Fanuc TP program (LS listing): ultrahose2.ls

/PROG  ultrahose2
/ATTR
COMMENT	= "19-03-19 19:07:18";
PROG_SIZE	= 0;
DEFAULT_GROUP	= 1, *, *, *, *;
/APPL
    ARC Welding Equipment: 1, *, *, *, *;
/MN
   1:  CALL HOME_ALL;
   1:  UFRAME_NUM = 1;
   1:  UTOOL_NUM = 3;
   1:  COL GUARD ADJUST 150;
   1:  PR[91] = PR[90];
   1:  PR[91,1] = PR[90,1] + -69.984;
   1:  PR[91,2] = PR[90,2] + 18.874;
   1:  PR[91,3] = PR[90,3] + 41.795;
   1:L PR[91] R[100]mm/sec CNT100;
   1:  PR[91,1] = PR[90,1] + -74.342;
   1:  PR[91,2] = PR[90,2] + 17.831;
   1:  PR[91,3] = PR[90,3] + 40.507;
   1:L PR[91] R[100]mm/sec CNT100;
   1:  PR[91,1] = PR[90,1] + -76.453;
   1:  PR[91,2] = PR[90,2] + 16.884;
   1:  PR[91,3] = PR[90,3] + 40.519;
   1:L PR[91] R[100]mm/sec CNT100;
   1:  PR[91,1] = PR[90,1] + -78.325;
   1:  PR[91,2] = PR[90,2] + 16.024;
   1:  PR[91,3] = PR[90,3] + 40.526;
   1:L PR[91] R[100]mm/sec CNT100;
   1:  PR[91,1] = PR[90,1] + -81.808;
   1:  PR[91,2] = PR[90,2] + 13.533;
   1:  PR[91,3] = PR[90,3] + 40.531;
   1:L PR[91] R[100]mm/sec CNT100;
   1:  PR[91,1] = PR[90,1] + -84.645;
   1:  PR[91,2] = PR[90,2] + 10.479;
   1:  PR[91,3] = PR[90,3] + 40.543;
   1:L PR[91] R[100]mm/sec CNT100;
   1:  PR[91,1] = PR[90,1] + -86.743;
   1:  PR[91,2] = PR[90,2] + 6.989;
   1:  PR[91,3] = PR[90,3] + 40.554;
   1:L PR[91] R[100]mm/sec CNT100;
   1:  PR[91,1] = PR[90,1] + -88.027;
   1:  PR[91,2] = PR[90,2] + 3.202;
   1:  PR[91,3] = PR[90,3] + 40.565;
   1:L PR[91] R[100]mm/sec CNT100;
   1:  PR[91,1] = PR[90,1] + -88.458;
   1:  PR[91,2] = PR[90,2] + -0.644;
   1:  PR[91,3] = PR[90,3] + 40.576;
   1:L PR[91] R[100]mm/sec CNT100;
   1:  PR[91,1] = PR[90,1] + -88.450;
   1:  PR[91,2] = PR[90,2] + -0.687;
   1:  PR[91,3] = PR[90,3] + 40.586;
   1:L PR[91] R[100]mm/sec CNT100;
   1:  PR[91,1] = PR[90,1] + -88.230;
   1:  PR[91,2] = PR[90,2] + -1.609;
   1:L PR[91] R[100]mm/sec CNT100;
   1:  PR[91,1] = PR[90,1] + -87.903;
   1:  PR[91,2] = PR[90,2] + -4.678;
   1:  PR[91,3] = PR[90,3] + 40.589;
   1:L PR[91] R[100]mm/sec CNT100;
   1:  PR[91,1] = PR[90,1] + -86.648;
   1:  PR[91,2] = PR[90,2] + -8.471;
   1:  PR[91,3] = PR[90,3] + 40.597;
   1:L PR[91] R[100]mm/sec CNT100;
   1:  PR[91,1] = PR[90,1] + -84.603;
   1:  PR[91,2] = PR[90,2] + -11.959;
   1:  PR[91,3] = PR[90,3] + 40.608;
   1:L PR[91] R[100]mm/sec CNT100;
   1:  PR[91,1] = PR[90,1] + -81.844;
   1:  PR[91,2] = PR[90,2] + -15.001;
   1:  PR[91,3] = PR[90,3] + 40.619;
   1:L PR[91] R[100]mm/sec CNT100;
   1:  PR[91,1] = PR[90,1] + -79.437;
   1:  PR[91,2] = PR[90,2] + -16.759;
   1:  PR[91,3] = PR[90,3] + 40.630;
   1:L PR[91] R[100]mm/sec CNT100;
   1:  PR[91,1] = PR[90,1] + -78.444;
   1:  PR[91,2] = PR[90,2] + -17.461;
   1:  PR[91,3] = PR[90,3] + 40.638;
   1:L PR[91] R[100]mm/sec CNT100;
   1:  PR[91,1] = PR[90,1] + -74.380;
   1:  PR[91,2] = PR[90,2] + -19.282;
   1:  PR[91,3] = PR[90,3] + 40.641;
   1:L PR[91] R[100]mm/sec CNT100;
   1:  PR[91,1] = PR[90,1] + -71.242;
   1:  PR[91,2] = PR[90,2] + -20.012;
   1:  PR[91,3] = PR[90,3] + 40.653;
   1:L PR[91] R[100]mm/sec CNT100;
   1:  PR[91,1] = PR[90,1] + -69.927;
   1:  PR[91,2] = PR[90,2] + -20.339;
   1:  PR[91,3] = PR[90,3] + 40.662;
   1:L PR[91] R[100]mm/sec CNT100;
   1:  PR[91,1] = PR[90,1] + -67.497;
   1:  PR[91,2] = PR[90,2] + -20.438;
   1:  PR[91,3] = PR[90,3] + 40.666;
   1:L PR[91] R[100]mm/sec CNT100;
   1:  PR[91,1] = PR[90,1] + -65.288;
   1:  PR[91,2] = PR[90,2] + -20.565;
   1:  PR[91,3] = PR[90,3] + 40.672;
   1:L PR[91] R[100]mm/sec CNT100;
   1:  PR[91,1] = PR[90,1] + -63.772;
   1:  PR[91,2] = PR[90,2] + -20.339;
   1:  PR[91,3] = PR[90,3] + 40.678;
   1:L PR[91] R[100]mm/sec CNT100;
   1:  PR[91,1] = PR[90,1] + -60.637;
   1:  PR[91,2] = PR[90,2] + -19.928;
   1:  PR[91,3] = PR[90,3] + 40.683;
   1:L PR[91] R[100]mm/sec CNT100;
   1:  PR[91,1] = PR[90,1] + -60.136;
   1:  PR[91,2] = PR[90,2] + -19.751;
   1:  PR[91,3] = PR[90,3] + 40.691;
   1:L PR[91] R[100]mm/sec CNT100;
   1:  PR[91,1] = PR[90,1] + -57.404;
   1:  PR[91,2] = PR[90,2] + -18.836;
   1:  PR[91,3] = PR[90,3] + 40.692;
   1:L PR[91] R[100]mm/sec CNT100;
   1:  PR[91,1] = PR[90,1] + -56.091;
   1:  PR[91,2] = PR[90,2] + -18.448;
   1:  PR[91,3] = PR[90,3] + 40.700;
   1:L PR[91] R[100]mm/sec CNT100;
   1:  PR[91,1] = PR[90,1] + -55.744;
   1:  PR[91,2] = PR[90,2] + -18.304;
   1:  PR[91,3] = PR[90,3] + 40.704;
   1:L PR[91] R[100]mm/sec CNT100;
   1:  PR[91,1] = PR[90,1] + -52.168;
   1:  PR[91,2] = PR[90,2] + -16.450;
   1:  PR[91,3] = PR[90,3] + 40.705;
   1:L PR[91] R[100]mm/sec CNT100;
   1:  PR[91,1] = PR[90,1] + -50.349;
   1:  PR[91,2] = PR[90,2] + -15.196;
   1:  PR[91,3] = PR[90,3] + 40.716;
   1:L PR[91] R[100]mm/sec CNT100;
   1:  PR[91,1] = PR[90,1] + -48.605;
   1:  PR[91,2] = PR[90,2] + -13.769;
   1:  PR[91,3] = PR[90,3] + 40.722;
   1:L PR[91] R[100]mm/sec CNT100;
   1:  PR[91,1] = PR[90,1] + -46.020;
   1:  PR[91,2] = PR[90,2] + -10.909;
   1:  PR[91,3] = PR[90,3] + 40.728;
   1:L PR[91] R[100]mm/sec CNT100;
   1:  PR[91,1] = PR[90,1] + -45.612;
   1:  PR[91,2] = PR[90,2] + -10.381;
   1:  PR[91,3] = PR[90,3] + 40.738;
   1:L PR[91] R[100]mm/sec CNT100;
   1:  PR[91,1] = PR[90,1] + -43.653;
   1:  PR[91,2] = PR[90,2] + -6.601;
   1:  PR[91,3] = PR[90,3] + 40.740;
   1:L PR[91] R[100]mm/sec CNT100;
   1:  PR[91,1] = PR[90,1] + -41.214;
   1:  PR[91,2] = PR[90,2] + -2.508;
   1:  PR[91,3] = PR[90,3] + 40.752;
   1:L PR[91] R[100]mm/sec CNT100;
   1:  PR[91,1] = PR[90,1] + -38.826;
   1:  PR[91,2] = PR[90,2] + -8.659;
   1:  PR[91,3] = PR[90,3] + 40.765;
   1:L PR[91] R[100]mm/sec CNT100;
   1:  PR[91,1] = PR[90,1] + -38.172;
   1:  PR[91,2] = PR[90,2] + -9.871;
   1:  PR[91,3] = PR[90,3] + 40.782;
   1:L PR[91] R[100]mm/sec CNT100;
   1:  PR[91,1] = PR[90,1] + -36.807;
   1:  PR[91,2] = PR[90,2] + -12.023;
   1:  PR[91,3] = PR[90,3] + 40.786;
   1:L PR[91] R[100]mm/sec CNT100;
   1:  PR[91,1] = PR[90,1] + -36.440;
   1:  PR[91,2] = PR[90,2] + -12.526;
   1:  PR[91,3] = PR[90,3] + 40.793;
   1:L PR[91] R[100]mm/sec CNT100;
   1:  PR[91,1] = PR[90,1] + -35.020;
   1:  PR[91,2] = PR[90,2] + -14.098;
   1:  PR[91,3] = PR[90,3] + 40.795;
   1:L PR[91] R[100]mm/sec CNT100;
   1:  PR[91,1] = PR[90,1] + -33.375;
   1:  PR[91,2] = PR[90,2] + -15.749;
   1:  PR[91,3] = PR[90,3] + 40.800;
   1:L PR[91] R[100]mm/sec CNT100;
   1:  PR[91,1] = PR[90,1] + -31.415;
   1:  PR[91,2] = PR[90,2] + -17.146;
   1:  PR[91,3] = PR[90,3] + 40.807;
   1:L PR[91] R[100]mm/sec CNT100;
   1:  PR[91,1] = PR[90,1] + -29.729;
   1:  PR[91,2] = PR[90,2] + -18.223;
   1:  PR[91,3] = PR[90,3] + 40.813;
   1:L PR[91] R[100]mm/sec CNT100;
   1:  PR[91,1] = PR[90,1] + -27.094;
   1:  PR[91,2] = PR[90,2] + -19.351;
   1:  PR[91,3] = PR[90,3] + 40.819;
   1:L PR[91] R[100]mm/sec CNT100;
   1:  PR[91,1] = PR[90,1] + -25.614;
   1:  PR[91,2] = PR[90,2] + -19.892;
   1:  PR[91,3] = PR[90,3] + 40.826;
   1:L PR[91] R[100]mm/sec CNT100;
   1:  PR[91,1] = PR[90,1] + -22.266;
   1:  PR[91,2] = PR[90,2] + -20.539;
   1:  PR[91,3] = PR[90,3] + 40.831;
   1:L PR[91] R[100]mm/sec CNT100;
   1:  PR[91,1] = PR[90,1] + -21.213;
   1:  PR[91,2] = PR[90,2] + -20.681;
   1:  PR[91,3] = PR[90,3] + 40.840;
   1:L PR[91] R[100]mm/sec CNT100;
   1:  PR[91,1] = PR[90,1] + -17.203;
   1:  PR[91,2] = PR[90,2] + -20.585;
   1:  PR[91,3] = PR[90,3] + 40.843;
   1:L PR[91] R[100]mm/sec CNT100;
   1:  PR[91,1] = PR[90,1] + -16.723;
   1:  PR[91,2] = PR[90,2] + -20.545;
   1:  PR[91,3] = PR[90,3] + 40.853;
   1:L PR[91] R[100]mm/sec CNT100;
   1:  PR[91,1] = PR[90,1] + -12.288;
   1:  PR[91,2] = PR[90,2] + -19.457;
   1:  PR[91,3] = PR[90,3] + 40.855;
   1:L PR[91] R[100]mm/sec CNT100;
   1:  PR[91,1] = PR[90,1] + -11.843;
   1:  PR[91,2] = PR[90,2] + -19.237;
   1:  PR[91,3] = PR[90,3] + 40.867;
   1:L PR[91] R[100]mm/sec CNT100;
   1:  PR[91,1] = PR[90,1] + -8.024;
   1:  PR[91,2] = PR[90,2] + -17.468;
   1:  PR[91,3] = PR[90,3] + 40.868;
   1:L PR[91] R[100]mm/sec CNT100;
   1:  PR[91,1] = PR[90,1] + -7.652;
   1:  PR[91,2] = PR[90,2] + -17.222;
   1:  PR[91,3] = PR[90,3] + 40.880;
   1:L PR[91] R[100]mm/sec CNT100;
   1:  PR[91,1] = PR[90,1] + -4.356;
   1:  PR[91,2] = PR[90,2] + -14.690;
   1:  PR[91,3] = PR[90,3] + 40.881;
   1:L PR[91] R[100]mm/sec CNT100;
   1:  PR[91,1] = PR[90,1] + -3.570;
   1:  PR[91,2] = PR[90,2] + -13.848;
   1:  PR[91,3] = PR[90,3] + 40.892;
   1:L PR[91] R[100]mm/sec CNT100;
   1:  PR[91,1] = PR[90,1] + -1.393;
   1:  PR[91,2] = PR[90,2] + -11.178;
   1:  PR[91,3] = PR[90,3] + 40.895;
   1:L PR[91] R[100]mm/sec CNT100;
   1:  PR[91,1] = PR[90,1] + -0.641;
   1:  PR[91,2] = PR[90,2] + -9.753;
   1:  PR[91,3] = PR[90,3] + 40.905;
   1:L PR[91] R[100]mm/sec CNT100;
   1:  PR[91,1] = PR[90,1] + 0.012;
   1:  PR[91,2] = PR[90,2] + -8.375;
   1:  PR[91,3] = PR[90,3] + 40.909;
   1:L PR[91] R[100]mm/sec CNT100;
   1:  PR[91,1] = PR[90,1] + 2.040;
   1:  PR[91,2] = PR[90,2] + -2.988;
   1:  PR[91,3] = PR[90,3] + 40.913;
   1:L PR[91] R[100]mm/sec CNT100;
   1:  PR[91,1] = PR[90,1] + 4.720;
   1:  PR[91,2] = PR[90,2] + -9.678;
   1:  PR[91,3] = PR[90,3] + 40.929;
   1:L PR[91] R[100]mm/sec CNT100;
   1:  PR[91,1] = PR[90,1] + 5.572;
   1:  PR[91,2] = PR[90,2] + -11.376;
   1:  PR[91,3] = PR[90,3] + 40.948;
   1:L PR[91] R[100]mm/sec CNT100;
   1:  PR[91,1] = PR[90,1] + 7.346;
   1:  PR[91,2] = PR[90,2] + -13.668;
   1:  PR[91,3] = PR[90,3] + 40.953;
   1:L PR[91] R[100]mm/sec CNT100;
   1:  PR[91,1] = PR[90,1] + 7.981;
   1:  PR[91,2] = PR[90,2] + -14.582;
   1:  PR[91,3] = PR[90,3] + 40.961;
   1:L PR[91] R[100]mm/sec CNT100;
   1:  PR[91,1] = PR[90,1] + 9.322;
   1:  PR[91,2] = PR[90,2] + -15.995;
   1:  PR[91,3] = PR[90,3] + 40.964;
   1:L PR[91] R[100]mm/sec CNT100;
   1:  PR[91,1] = PR[90,1] + 12.105;
   1:  PR[91,2] = PR[90,2] + -18.105;
   1:  PR[91,3] = PR[90,3] + 40.969;
   1:L PR[91] R[100]mm/sec CNT100;
   1:  PR[91,1] = PR[90,1] + 13.658;
   1:  PR[91,2] = PR[90,2] + -19.073;
   1:  PR[91,3] = PR[90,3] + 40.979;
   1:L PR[91] R[100]mm/sec CNT100;
   1:  PR[91,1] = PR[90,1] + 17.034;
   1:  PR[91,2] = PR[90,2] + -20.451;
   1:  PR[91,3] = PR[90,3] + 40.984;
   1:L PR[91] R[100]mm/sec CNT100;
   1:  PR[91,1] = PR[90,1] + 18.629;
   1:  PR[91,2] = PR[90,2] + -20.956;
   1:  PR[91,3] = PR[90,3] + 40.994;
   1:L PR[91] R[100]mm/sec CNT100;
   1:  PR[91,1] = PR[90,1] + 22.409;
   1:  PR[91,2] = PR[90,2] + -21.441;
   1:  PR[91,3] = PR[90,3] + 40.998;
   1:L PR[91] R[100]mm/sec CNT100;
   1:  PR[91,1] = PR[90,1] + 23.913;
   1:  PR[91,2] = PR[90,2] + -21.527;
   1:  PR[91,3] = PR[90,3] + 41.008;
   1:L PR[91] R[100]mm/sec CNT100;
   1:  PR[91,1] = PR[90,1] + 27.852;
   1:  PR[91,2] = PR[90,2] + -21.002;
   1:  PR[91,3] = PR[90,3] + 41.012;
   1:L PR[91] R[100]mm/sec CNT100;
   1:  PR[91,1] = PR[90,1] + 29.169;
   1:  PR[91,2] = PR[90,2] + -20.747;
   1:  PR[91,3] = PR[90,3] + 41.023;
   1:L PR[91] R[100]mm/sec CNT100;
   1:  PR[91,1] = PR[90,1] + 32.982;
   1:  PR[91,2] = PR[90,2] + -19.175;
   1:  PR[91,3] = PR[90,3] + 41.027;
   1:L PR[91] R[100]mm/sec CNT100;
   1:  PR[91,1] = PR[90,1] + 34.056;
   1:  PR[91,2] = PR[90,2] + -18.671;
   1:  PR[91,3] = PR[90,3] + 41.038;
   1:L PR[91] R[100]mm/sec CNT100;
   1:  PR[91,1] = PR[90,1] + 37.540;
   1:  PR[91,2] = PR[90,2] + -16.026;
   1:  PR[91,3] = PR[90,3] + 41.041;
   1:L PR[91] R[100]mm/sec CNT100;
   1:  PR[91,1] = PR[90,1] + 37.772;
   1:  PR[91,2] = PR[90,2] + -15.879;
   1:  PR[91,3] = PR[90,3] + 41.053;
   1:L PR[91] R[100]mm/sec CNT100;
   1:  PR[91,1] = PR[90,1] + 38.445;
   1:  PR[91,2] = PR[90,2] + -15.255;
   1:  PR[91,3] = PR[90,3] + 41.054;
   1:L PR[91] R[100]mm/sec CNT100;
   1:  PR[91,1] = PR[90,1] + 38.894;
   1:  PR[91,2] = PR[90,2] + -14.763;
   1:  PR[91,3] = PR[90,3] + 41.056;
   1:L PR[91] R[100]mm/sec CNT100;
   1:  PR[91,1] = PR[90,1] + 41.536;
   1:  PR[91,2] = PR[90,2] + -11.574;
   1:  PR[91,3] = PR[90,3] + 41.058;
   1:L PR[91] R[100]mm/sec CNT100;
   1:  PR[91,1] = PR[90,1] + 44.233;
   1:  PR[91,2] = PR[90,2] + -14.310;
   1:  PR[91,3] = PR[90,3] + 41.069;
   1:L PR[91] R[100]mm/sec CNT100;
   1:  PR[91,1] = PR[90,1] + 46.319;
   1:  PR[91,2] = PR[90,2] + -15.800;
   1:  PR[91,3] = PR[90,3] + 41.080;
   1:L PR[91] R[100]mm/sec CNT100;
   1:  PR[91,1] = PR[90,1] + 49.840;
   1:  PR[91,2] = PR[90,2] + -18.103;
   1:  PR[91,3] = PR[90,3] + 41.086;
   1:L PR[91] R[100]mm/sec CNT100;
   1:  PR[91,1] = PR[90,1] + 50.344;
   1:  PR[91,2] = PR[90,2] + -18.304;
   1:  PR[91,3] = PR[90,3] + 41.098;
   1:L PR[91] R[100]mm/sec CNT100;
   1:  PR[91,1] = PR[90,1] + 54.403;
   1:  PR[91,2] = PR[90,2] + -20.079;
   1:  PR[91,3] = PR[90,3] + 41.099;
   1:L PR[91] R[100]mm/sec CNT100;
   1:  PR[91,1] = PR[90,1] + 56.501;
   1:  PR[91,2] = PR[90,2] + -20.784;
   1:  PR[91,3] = PR[90,3] + 41.111;
   1:L PR[91] R[100]mm/sec CNT100;
   1:  PR[91,1] = PR[90,1] + 59.032;
   1:  PR[91,2] = PR[90,2] + -21.322;
   1:  PR[91,3] = PR[90,3] + 41.117;
   1:L PR[91] R[100]mm/sec CNT100;
   1:  PR[91,1] = PR[90,1] + 63.968;
   1:  PR[91,2] = PR[90,2] + -21.878;
   1:  PR[91,3] = PR[90,3] + 41.124;
   1:L PR[91] R[100]mm/sec CNT100;
   1:  PR[91,1] = PR[90,1] + 64.084;
   1:  PR[91,2] = PR[90,2] + -21.880;
   1:  PR[91,3] = PR[90,3] + 41.138;
   1:L PR[91] R[100]mm/sec CNT100;
   1:  PR[91,1] = PR[90,1] + 64.736;
   1:  PR[91,2] = PR[90,2] + -21.820;
   1:L PR[91] R[100]mm/sec CNT100;
   1:  PR[91,1] = PR[90,1] + 69.228;
   1:  PR[91,2] = PR[90,2] + -21.507;
   1:  PR[91,3] = PR[90,3] + 41.140;
   1:L PR[91] R[100]mm/sec CNT100;
   1:  PR[91,1] = PR[90,1] + 70.397;
   1:  PR[91,2] = PR[90,2] + -21.313;
   1:  PR[91,3] = PR[90,3] + 41.152;
   1:L PR[91] R[100]mm/sec CNT100;
   1:  PR[91,1] = PR[90,1] + 73.749;
   1:  PR[91,2] = PR[90,2] + -20.328;
   1:  PR[91,3] = PR[90,3] + 41.155;
   1:L PR[91] R[100]mm/sec CNT100;
   1:  PR[91,1] = PR[90,1] + 75.998;
   1:  PR[91,2] = PR[90,2] + -19.468;
   1:  PR[91,3] = PR[90,3] + 41.164;
   1:L PR[91] R[100]mm/sec CNT100;
   1:  PR[91,1] = PR[90,1] + 77.841;
   1:  PR[91,2] = PR[90,2] + -18.450;
   1:  PR[91,3] = PR[90,3] + 41.171;
   1:L PR[91] R[100]mm/sec CNT100;
   1:  PR[91,1] = PR[90,1] + 80.605;
   1:  PR[91,2] = PR[90,2] + -16.678;
   1:  PR[91,3] = PR[90,3] + 41.177;
   1:L PR[91] R[100]mm/sec CNT100;
   1:  PR[91,1] = PR[90,1] + 81.422;
   1:  PR[91,2] = PR[90,2] + -15.949;
   1:  PR[91,3] = PR[90,3] + 41.186;
   1:L PR[91] R[100]mm/sec CNT100;
   1:  PR[91,1] = PR[90,1] + 84.184;
   1:  PR[91,2] = PR[90,2] + -13.215;
   1:  PR[91,3] = PR[90,3] + 41.189;
   1:L PR[91] R[100]mm/sec CNT100;
   1:  PR[91,1] = PR[90,1] + 84.403;
   1:  PR[91,2] = PR[90,2] + -12.900;
   1:  PR[91,3] = PR[90,3] + 41.199;
   1:L PR[91] R[100]mm/sec CNT100;
   1:  PR[91,1] = PR[90,1] + 86.719;
   1:  PR[91,2] = PR[90,2] + -9.308;
   1:  PR[91,3] = PR[90,3] + 41.200;
   1:L PR[91] R[100]mm/sec CNT100;
   1:  PR[91,1] = PR[90,1] + 87.451;
   1:  PR[91,2] = PR[90,2] + -7.293;
   1:  PR[91,3] = PR[90,3] + 41.212;
   1:L PR[91] R[100]mm/sec CNT100;
   1:  PR[91,1] = PR[90,1] + 88.212;
   1:  PR[91,2] = PR[90,2] + -5.114;
   1:  PR[91,3] = PR[90,3] + 41.217;
   1:L PR[91] R[100]mm/sec CNT100;
   1:  PR[91,1] = PR[90,1] + 88.706;
   1:  PR[91,2] = PR[90,2] + -0.729;
   1:  PR[91,3] = PR[90,3] + 41.224;
   1:L PR[91] R[100]mm/sec CNT100;
   1:  PR[91,1] = PR[90,1] + 88.212;
   1:  PR[91,2] = PR[90,2] + 3.655;
   1:  PR[91,3] = PR[90,3] + 41.236;
   1:L PR[91] R[100]mm/sec CNT100;
   1:  PR[91,1] = PR[90,1] + 87.451;
   1:  PR[91,2] = PR[90,2] + 5.834;
   1:  PR[91,3] = PR[90,3] + 41.247;
   1:L PR[91] R[100]mm/sec CNT100;
   1:  PR[91,1] = PR[90,1] + 86.719;
   1:  PR[91,2] = PR[90,2] + 7.849;
   1:  PR[91,3] = PR[90,3] + 41.254;
   1:L PR[91] R[100]mm/sec CNT100;
   1:  PR[91,1] = PR[90,1] + 84.403;
   1:  PR[91,2] = PR[90,2] + 11.441;
   1:  PR[91,3] = PR[90,3] + 41.259;
   1:L PR[91] R[100]mm/sec CNT100;
   1:  PR[91,1] = PR[90,1] + 84.184;
   1:  PR[91,2] = PR[90,2] + 11.756;
   1:  PR[91,3] = PR[90,3] + 41.271;
   1:L PR[91] R[100]mm/sec CNT100;
   1:  PR[91,1] = PR[90,1] + 81.422;
   1:  PR[91,2] = PR[90,2] + 14.490;
   1:  PR[91,3] = PR[90,3] + 41.272;
   1:L PR[91] R[100]mm/sec CNT100;
   1:  PR[91,1] = PR[90,1] + 80.605;
   1:  PR[91,2] = PR[90,2] + 15.219;
   1:  PR[91,3] = PR[90,3] + 41.283;
   1:L PR[91] R[100]mm/sec CNT100;
   1:  PR[91,1] = PR[90,1] + 77.841;
   1:  PR[91,2] = PR[90,2] + 16.991;
   1:  PR[91,3] = PR[90,3] + 41.285;
   1:L PR[91] R[100]mm/sec CNT100;
   1:  PR[91,1] = PR[90,1] + 75.998;
   1:  PR[91,2] = PR[90,2] + 18.009;
   1:  PR[91,3] = PR[90,3] + 41.294;
   1:L PR[91] R[100]mm/sec CNT100;
   1:  PR[91,1] = PR[90,1] + 73.749;
   1:  PR[91,2] = PR[90,2] + 18.869;
   1:  PR[91,3] = PR[90,3] + 41.300;
   1:L PR[91] R[100]mm/sec CNT100;
   1:  PR[91,1] = PR[90,1] + 70.398;
   1:  PR[91,2] = PR[90,2] + 19.854;
   1:  PR[91,3] = PR[90,3] + 41.307;
   1:L PR[91] R[100]mm/sec CNT100;
   1:  PR[91,1] = PR[90,1] + 69.229;
   1:  PR[91,2] = PR[90,2] + 20.048;
   1:  PR[91,3] = PR[90,3] + 41.316;
   1:L PR[91] R[100]mm/sec CNT100;
   1:  PR[91,1] = PR[90,1] + 64.736;
   1:  PR[91,2] = PR[90,2] + 20.362;
   1:  PR[91,3] = PR[90,3] + 41.319;
   1:L PR[91] R[100]mm/sec CNT100;
   1:  PR[91,1] = PR[90,1] + 64.085;
   1:  PR[91,2] = PR[90,2] + 20.421;
   1:  PR[91,3] = PR[90,3] + 41.331;
   1:L PR[91] R[100]mm/sec CNT100;
   1:  PR[91,1] = PR[90,1] + 63.965;
   1:  PR[91,2] = PR[90,2] + 20.419;
   1:  PR[91,3] = PR[90,3] + 41.333;
   1:L PR[91] R[100]mm/sec CNT100;
   1:  PR[91,1] = PR[90,1] + 59.012;
   1:  PR[91,2] = PR[90,2] + 19.862;
   1:L PR[91] R[100]mm/sec CNT100;
   1:  PR[91,1] = PR[90,1] + 56.444;
   1:  PR[91,2] = PR[90,2] + 19.308;
   1:  PR[91,3] = PR[90,3] + 41.347;
   1:L PR[91] R[100]mm/sec CNT100;
   1:  PR[91,1] = PR[90,1] + 54.358;
   1:  PR[91,2] = PR[90,2] + 18.607;
   1:  PR[91,3] = PR[90,3] + 41.354;
   1:L PR[91] R[100]mm/sec CNT100;
   1:  PR[91,1] = PR[90,1] + 50.348;
   1:  PR[91,2] = PR[90,2] + 16.837;
   1:  PR[91,3] = PR[90,3] + 41.360;
   1:L PR[91] R[100]mm/sec CNT100;
   1:  PR[91,1] = PR[90,1] + 49.750;
   1:  PR[91,2] = PR[90,2] + 16.598;
   1:  PR[91,3] = PR[90,3] + 41.372;
   1:L PR[91] R[100]mm/sec CNT100;
   1:  PR[91,1] = PR[90,1] + 46.292;
   1:  PR[91,2] = PR[90,2] + 14.311;
   1:  PR[91,3] = PR[90,3] + 41.374;
   1:L PR[91] R[100]mm/sec CNT100;
   1:  PR[91,1] = PR[90,1] + 44.217;
   1:  PR[91,2] = PR[90,2] + 12.836;
   1:  PR[91,3] = PR[90,3] + 41.385;
   1:L PR[91] R[100]mm/sec CNT100;
   1:  PR[91,1] = PR[90,1] + 41.504;
   1:  PR[91,2] = PR[90,2] + 9.965;
   1:  PR[91,3] = PR[90,3] + 41.392;
   1:L PR[91] R[100]mm/sec CNT100;
   1:  PR[91,1] = PR[90,1] + 38.885;
   1:  PR[91,2] = PR[90,2] + 13.307;
   1:  PR[91,3] = PR[90,3] + 41.402;
   1:L PR[91] R[100]mm/sec CNT100;
   1:  PR[91,1] = PR[90,1] + 37.659;
   1:  PR[91,2] = PR[90,2] + 14.522;
   1:  PR[91,3] = PR[90,3] + 41.414;
   1:L PR[91] R[100]mm/sec CNT100;
   1:  PR[91,1] = PR[90,1] + 34.585;
   1:  PR[91,2] = PR[90,2] + 16.847;
   1:  PR[91,3] = PR[90,3] + 41.418;
   1:L PR[91] R[100]mm/sec CNT100;
   1:  PR[91,1] = PR[90,1] + 34.176;
   1:  PR[91,2] = PR[90,2] + 17.142;
   1:  PR[91,3] = PR[90,3] + 41.429;
   1:L PR[91] R[100]mm/sec CNT100;
   1:  PR[91,1] = PR[90,1] + 34.085;
   1:  PR[91,2] = PR[90,2] + 17.201;
   1:  PR[91,3] = PR[90,3] + 41.430;
   1:L PR[91] R[100]mm/sec CNT100;
   1:  PR[91,1] = PR[90,1] + 32.952;
   1:  PR[91,2] = PR[90,2] + 17.734;
   1:L PR[91] R[100]mm/sec CNT100;
   1:  PR[91,1] = PR[90,1] + 29.141;
   1:  PR[91,2] = PR[90,2] + 19.296;
   1:  PR[91,3] = PR[90,3] + 41.434;
   1:L PR[91] R[100]mm/sec CNT100;
   1:  PR[91,1] = PR[90,1] + 27.825;
   1:  PR[91,2] = PR[90,2] + 19.551;
   1:  PR[91,3] = PR[90,3] + 41.445;
   1:L PR[91] R[100]mm/sec CNT100;
   1:  PR[91,1] = PR[90,1] + 23.890;
   1:  PR[91,2] = PR[90,2] + 20.068;
   1:  PR[91,3] = PR[90,3] + 41.449;
   1:L PR[91] R[100]mm/sec CNT100;
   1:  PR[91,1] = PR[90,1] + 22.387;
   1:  PR[91,2] = PR[90,2] + 19.982;
   1:  PR[91,3] = PR[90,3] + 41.459;
   1:L PR[91] R[100]mm/sec CNT100;
   1:  PR[91,1] = PR[90,1] + 18.613;
   1:  PR[91,2] = PR[90,2] + 19.493;
   1:  PR[91,3] = PR[90,3] + 41.463;
   1:L PR[91] R[100]mm/sec CNT100;
   1:  PR[91,1] = PR[90,1] + 17.018;
   1:  PR[91,2] = PR[90,2] + 18.989;
   1:  PR[91,3] = PR[90,3] + 41.474;
   1:L PR[91] R[100]mm/sec CNT100;
   1:  PR[91,1] = PR[90,1] + 13.648;
   1:  PR[91,2] = PR[90,2] + 17.609;
   1:  PR[91,3] = PR[90,3] + 41.478;
   1:L PR[91] R[100]mm/sec CNT100;
   1:  PR[91,1] = PR[90,1] + 12.096;
   1:  PR[91,2] = PR[90,2] + 16.642;
   1:  PR[91,3] = PR[90,3] + 41.488;
   1:L PR[91] R[100]mm/sec CNT100;
   1:  PR[91,1] = PR[90,1] + 9.318;
   1:  PR[91,2] = PR[90,2] + 14.532;
   1:  PR[91,3] = PR[90,3] + 41.493;
   1:L PR[91] R[100]mm/sec CNT100;
   1:  PR[91,1] = PR[90,1] + 7.941;
   1:  PR[91,2] = PR[90,2] + 13.084;
   1:  PR[91,3] = PR[90,3] + 41.502;
   1:L PR[91] R[100]mm/sec CNT100;
   1:  PR[91,1] = PR[90,1] + 5.848;
   1:  PR[91,2] = PR[90,2] + 10.378;
   1:  PR[91,3] = PR[90,3] + 41.508;
   1:L PR[91] R[100]mm/sec CNT100;
   1:  PR[91,1] = PR[90,1] + 5.791;
   1:  PR[91,2] = PR[90,2] + 10.293;
   1:  PR[91,3] = PR[90,3] + 41.517;
   1:L PR[91] R[100]mm/sec CNT100;
   1:  PR[91,1] = PR[90,1] + 5.693;
   1:  PR[91,2] = PR[90,2] + 10.137;
   1:L PR[91] R[100]mm/sec CNT100;
   1:  PR[91,1] = PR[90,1] + 4.942;
   1:  PR[91,2] = PR[90,2] + 8.700;
   1:  PR[91,3] = PR[90,3] + 41.518;
   1:L PR[91] R[100]mm/sec CNT100;
   1:  PR[91,1] = PR[90,1] + 4.314;
   1:  PR[91,2] = PR[90,2] + 7.197;
   1:  PR[91,3] = PR[90,3] + 41.522;
   1:L PR[91] R[100]mm/sec CNT100;
   1:  PR[91,1] = PR[90,1] + 2.218;
   1:  PR[91,2] = PR[90,2] + 1.901;
   1:  PR[91,3] = PR[90,3] + 41.527;
   1:L PR[91] R[100]mm/sec CNT100;
   1:  PR[91,1] = PR[90,1] + -0.867;
   1:  PR[91,2] = PR[90,2] + 8.750;
   1:  PR[91,3] = PR[90,3] + 41.542;
   1:L PR[91] R[100]mm/sec CNT100;
   1:  PR[91,1] = PR[90,1] + -1.376;
   1:  PR[91,2] = PR[90,2] + 9.695;
   1:  PR[91,3] = PR[90,3] + 41.562;
   1:L PR[91] R[100]mm/sec CNT100;
   1:  PR[91,1] = PR[90,1] + -3.553;
   1:  PR[91,2] = PR[90,2] + 12.368;
   1:  PR[91,3] = PR[90,3] + 41.565;
   1:L PR[91] R[100]mm/sec CNT100;
   1:  PR[91,1] = PR[90,1] + -4.343;
   1:  PR[91,2] = PR[90,2] + 13.219;
   1:  PR[91,3] = PR[90,3] + 41.574;
   1:L PR[91] R[100]mm/sec CNT100;
   1:  PR[91,1] = PR[90,1] + -7.635;
   1:  PR[91,2] = PR[90,2] + 15.753;
   1:  PR[91,3] = PR[90,3] + 41.578;
   1:L PR[91] R[100]mm/sec CNT100;
   1:  PR[91,1] = PR[90,1] + -8.010;
   1:  PR[91,2] = PR[90,2] + 16.001;
   1:  PR[91,3] = PR[90,3] + 41.589;
   1:L PR[91] R[100]mm/sec CNT100;
   1:  PR[91,1] = PR[90,1] + -11.844;
   1:  PR[91,2] = PR[90,2] + 17.780;
   1:  PR[91,3] = PR[90,3] + 41.590;
   1:L PR[91] R[100]mm/sec CNT100;
   1:  PR[91,1] = PR[90,1] + -12.274;
   1:  PR[91,2] = PR[90,2] + 17.993;
   1:  PR[91,3] = PR[90,3] + 41.601;
   1:L PR[91] R[100]mm/sec CNT100;
   1:  PR[91,1] = PR[90,1] + -16.710;
   1:  PR[91,2] = PR[90,2] + 19.085;
   1:  PR[91,3] = PR[90,3] + 41.603;
   1:L PR[91] R[100]mm/sec CNT100;
   1:  PR[91,1] = PR[90,1] + -17.189;
   1:  PR[91,2] = PR[90,2] + 19.124;
   1:  PR[91,3] = PR[90,3] + 41.615;
   1:L PR[91] R[100]mm/sec CNT100;
   1:  PR[91,1] = PR[90,1] + -21.203;
   1:  PR[91,2] = PR[90,2] + 19.223;
   1:  PR[91,3] = PR[90,3] + 41.616;
   1:L PR[91] R[100]mm/sec CNT100;
   1:  PR[91,1] = PR[90,1] + -22.255;
   1:  PR[91,2] = PR[90,2] + 19.081;
   1:  PR[91,3] = PR[90,3] + 41.627;
   1:L PR[91] R[100]mm/sec CNT100;
   1:  PR[91,1] = PR[90,1] + -25.606;
   1:  PR[91,2] = PR[90,2] + 18.436;
   1:  PR[91,3] = PR[90,3] + 41.630;
   1:L PR[91] R[100]mm/sec CNT100;
   1:  PR[91,1] = PR[90,1] + -27.085;
   1:  PR[91,2] = PR[90,2] + 17.895;
   1:  PR[91,3] = PR[90,3] + 41.639;
   1:L PR[91] R[100]mm/sec CNT100;
   1:  PR[91,1] = PR[90,1] + -29.723;
   1:  PR[91,2] = PR[90,2] + 16.767;
   1:  PR[91,3] = PR[90,3] + 41.644;
   1:L PR[91] R[100]mm/sec CNT100;
   1:  PR[91,1] = PR[90,1] + -31.409;
   1:  PR[91,2] = PR[90,2] + 15.691;
   1:  PR[91,3] = PR[90,3] + 41.651;
   1:L PR[91] R[100]mm/sec CNT100;
   1:  PR[91,1] = PR[90,1] + -33.371;
   1:  PR[91,2] = PR[90,2] + 14.294;
   1:  PR[91,3] = PR[90,3] + 41.657;
   1:L PR[91] R[100]mm/sec CNT100;
   1:  PR[91,1] = PR[90,1] + -35.015;
   1:  PR[91,2] = PR[90,2] + 12.643;
   1:  PR[91,3] = PR[90,3] + 41.663;
   1:L PR[91] R[100]mm/sec CNT100;
   1:  PR[91,1] = PR[90,1] + -36.390;
   1:  PR[91,2] = PR[90,2] + 11.125;
   1:  PR[91,3] = PR[90,3] + 41.669;
   1:L PR[91] R[100]mm/sec CNT100;
   1:  PR[91,1] = PR[90,1] + -37.846;
   1:  PR[91,2] = PR[90,2] + 8.812;
   1:  PR[91,3] = PR[90,3] + 41.675;
   1:L PR[91] R[100]mm/sec CNT100;
   1:  PR[91,1] = PR[90,1] + -38.076;
   1:  PR[91,2] = PR[90,2] + 8.534;
   1:  PR[91,3] = PR[90,3] + 41.682;
   1:L PR[91] R[100]mm/sec CNT100;
   1:  PR[91,1] = PR[90,1] + -38.403;
   1:  PR[91,2] = PR[90,2] + 8.035;
   1:  PR[91,3] = PR[90,3] + 41.683;
   1:L PR[91] R[100]mm/sec CNT100;
   1:  PR[91,1] = PR[90,1] + -38.759;
   1:  PR[91,2] = PR[90,2] + 7.344;
   1:  PR[91,3] = PR[90,3] + 41.685;
   1:L PR[91] R[100]mm/sec CNT100;
   1:  PR[91,1] = PR[90,1] + -39.268;
   1:  PR[91,2] = PR[90,2] + 5.891;
   1:  PR[91,3] = PR[90,3] + 41.687;
   1:L PR[91] R[100]mm/sec CNT100;
   1:  PR[91,1] = PR[90,1] + -39.389;
   1:  PR[91,2] = PR[90,2] + 5.694;
   1:  PR[91,3] = PR[90,3] + 41.691;
   1:L PR[91] R[100]mm/sec CNT100;
   1:  PR[91,1] = PR[90,1] + -41.513;
   1:  PR[91,2] = PR[90,2] + 0.383;
   1:  PR[91,3] = PR[90,3] + 41.692;
   1:L PR[91] R[100]mm/sec CNT100;
   1:  PR[91,1] = PR[90,1] + -44.557;
   1:  PR[91,2] = PR[90,2] + 7.369;
   1:  PR[91,3] = PR[90,3] + 41.707;
   1:L PR[91] R[100]mm/sec CNT100;
   1:  PR[91,1] = PR[90,1] + -45.645;
   1:  PR[91,2] = PR[90,2] + 8.862;
   1:  PR[91,3] = PR[90,3] + 41.728;
   1:L PR[91] R[100]mm/sec CNT100;
   1:  PR[91,1] = PR[90,1] + -47.705;
   1:  PR[91,2] = PR[90,2] + 11.387;
   1:  PR[91,3] = PR[90,3] + 41.733;
   1:L PR[91] R[100]mm/sec CNT100;
   1:  PR[91,1] = PR[90,1] + -48.151;
   1:  PR[91,2] = PR[90,2] + 11.764;
   1:  PR[91,3] = PR[90,3] + 41.742;
   1:L PR[91] R[100]mm/sec CNT100;
   1:  PR[91,1] = PR[90,1] + -49.875;
   1:  PR[91,2] = PR[90,2] + 13.098;
   1:  PR[91,3] = PR[90,3] + 41.743;
   1:L PR[91] R[100]mm/sec CNT100;
   1:  PR[91,1] = PR[90,1] + -51.686;
   1:  PR[91,2] = PR[90,2] + 14.649;
   1:  PR[91,3] = PR[90,3] + 41.749;
   1:L PR[91] R[100]mm/sec CNT100;
   1:  PR[91,1] = PR[90,1] + -55.941;
   1:  PR[91,2] = PR[90,2] + 16.976;
   1:  PR[91,3] = PR[90,3] + 41.756;
   1:L PR[91] R[100]mm/sec CNT100;
   1:  PR[91,1] = PR[90,1] + -58.858;
   1:  PR[91,2] = PR[90,2] + 17.920;
   1:  PR[91,3] = PR[90,3] + 41.769;
   1:L PR[91] R[100]mm/sec CNT100;
   1:  PR[91,1] = PR[90,1] + -60.595;
   1:  PR[91,2] = PR[90,2] + 18.463;
   1:  PR[91,3] = PR[90,3] + 41.777;
   1:L PR[91] R[100]mm/sec CNT100;
   1:  PR[91,1] = PR[90,1] + -65.427;
   1:  PR[91,2] = PR[90,2] + 19.085;
   1:  PR[91,3] = PR[90,3] + 41.782;
   1:L PR[91] R[100]mm/sec CNT100;
   1:  PR[91] = PR[90];
   1:  PR[91,1] = PR[90,1] + -67.474;
   1:  PR[91,3] = PR[90,3] + 43.095;
   1:L PR[91] R[100]mm/sec CNT100;
   1:  PR[91,1] = PR[90,1] + -69.465;
   1:  PR[91,2] = PR[90,2] + 18.992;
   1:  PR[91,3] = PR[90,3] + 41.803;
   1:L PR[91] R[100]mm/sec CNT100;
   1:  PR[91,1] = PR[90,1] + -73.840;
   1:  PR[91,2] = PR[90,2] + 17.937;
   1:  PR[91,3] = PR[90,3] + 41.808;
   1:L PR[91] R[100]mm/sec CNT100;
   1:  PR[91,1] = PR[90,1] + -77.850;
   1:  PR[91,2] = PR[90,2] + 16.111;
   1:  PR[91,3] = PR[90,3] + 41.821;
   1:L PR[91] R[100]mm/sec CNT100;
   1:  PR[91,1] = PR[90,1] + -81.344;
   1:  PR[91,2] = PR[90,2] + 13.606;
   1:  PR[91,3] = PR[90,3] + 41.833;
   1:L PR[91] R[100]mm/sec CNT100;
   1:  PR[91,1] = PR[90,1] + -84.191;
   1:  PR[91,2] = PR[90,2] + 10.533;
   1:  PR[91,3] = PR[90,3] + 41.845;
   1:L PR[91] R[100]mm/sec CNT100;
   1:  PR[91,1] = PR[90,1] + -86.296;
   1:  PR[91,2] = PR[90,2] + 7.025;
   1:  PR[91,3] = PR[90,3] + 41.856;
   1:L PR[91] R[100]mm/sec CNT100;
   1:  PR[91,1] = PR[90,1] + -87.585;
   1:  PR[91,2] = PR[90,2] + 3.222;
   1:  PR[91,3] = PR[90,3] + 41.867;
   1:L PR[91] R[100]mm/sec CNT100;
   1:  PR[91,1] = PR[90,1] + -87.989;
   1:  PR[91,2] = PR[90,2] + -0.429;
   1:  PR[91,3] = PR[90,3] + 41.879;
   1:L PR[91] R[100]mm/sec CNT100;
   1:  PR[91,1] = PR[90,1] + -88.046;
   1:  PR[91,2] = PR[90,2] + -0.702;
   1:  PR[91,3] = PR[90,3] + 41.889;
   1:L PR[91] R[100]mm/sec CNT100;
   1:  PR[91,1] = PR[90,1] + -87.939;
   1:  PR[91,2] = PR[90,2] + -1.154;
   1:L PR[91] R[100]mm/sec CNT100;
   1:  PR[91,1] = PR[90,1] + -87.561;
   1:  PR[91,2] = PR[90,2] + -4.693;
   1:  PR[91,3] = PR[90,3] + 41.891;
   1:L PR[91] R[100]mm/sec CNT100;
   1:  PR[91,1] = PR[90,1] + -86.303;
   1:  PR[91,2] = PR[90,2] + -8.501;
   1:  PR[91,3] = PR[90,3] + 41.901;
   1:L PR[91] R[100]mm/sec CNT100;
   1:  PR[91,1] = PR[90,1] + -84.252;
   1:  PR[91,2] = PR[90,2] + -12.004;
   1:  PR[91,3] = PR[90,3] + 41.912;
   1:L PR[91] R[100]mm/sec CNT100;
   1:  PR[91,1] = PR[90,1] + -82.472;
   1:  PR[91,2] = PR[90,2] + -13.969;
   1:  PR[91,3] = PR[90,3] + 41.923;
   1:L PR[91] R[100]mm/sec CNT100;
   1:  PR[91,1] = PR[90,1] + -81.462;
   1:  PR[91,2] = PR[90,2] + -15.043;
   1:  PR[91,3] = PR[90,3] + 41.930;
   1:L PR[91] R[100]mm/sec CNT100;
   1:  PR[91,1] = PR[90,1] + -77.908;
   1:  PR[91,2] = PR[90,2] + -17.555;
   1:  PR[91,3] = PR[90,3] + 41.934;
   1:L PR[91] R[100]mm/sec CNT100;
   1:  PR[91,1] = PR[90,1] + -74.860;
   1:  PR[91,2] = PR[90,2] + -18.913;
   1:  PR[91,3] = PR[90,3] + 41.946;
   1:L PR[91] R[100]mm/sec CNT100;
   1:  PR[91,1] = PR[90,1] + -73.811;
   1:  PR[91,2] = PR[90,2] + -19.397;
   1:  PR[91,3] = PR[90,3] + 41.955;
   1:L PR[91] R[100]mm/sec CNT100;
   1:  PR[91,1] = PR[90,1] + -71.225;
   1:  PR[91,2] = PR[90,2] + -19.999;
   1:  PR[91,3] = PR[90,3] + 41.959;
   1:L PR[91] R[100]mm/sec CNT100;
   1:  PR[91,1] = PR[90,1] + -69.344;
   1:  PR[91,2] = PR[90,2] + -20.467;
   1:  PR[91,3] = PR[90,3] + 41.966;
   1:L PR[91] R[100]mm/sec CNT100;
   1:  PR[91,1] = PR[90,1] + -67.500;
   1:  PR[91,2] = PR[90,2] + -20.542;
   1:  PR[91,3] = PR[90,3] + 41.971;
   1:L PR[91] R[100]mm/sec CNT100;
   1:  PR[91,1] = PR[90,1] + -64.674;
   1:  PR[91,2] = PR[90,2] + -20.705;
   1:  PR[91,3] = PR[90,3] + 41.976;
   1:L PR[91] R[100]mm/sec CNT100;
   1:  PR[91,1] = PR[90,1] + -63.773;
   1:  PR[91,2] = PR[90,2] + -20.570;
   1:  PR[91,3] = PR[90,3] + 41.984;
   1:L PR[91] R[100]mm/sec CNT100;
   1:  PR[91,1] = PR[90,1] + -59.973;
   1:  PR[91,2] = PR[90,2] + -20.073;
   1:  PR[91,3] = PR[90,3] + 41.987;
   1:L PR[91] R[100]mm/sec CNT100;
   1:  PR[91,1] = PR[90,1] + -59.827;
   1:  PR[91,2] = PR[90,2] + -20.023;
   1:  PR[91,3] = PR[90,3] + 41.997;
   1:L PR[91] R[100]mm/sec CNT100;
   1:  PR[91,1] = PR[90,1] + -55.586;
   1:  PR[91,2] = PR[90,2] + -18.768;
   1:  PR[91,3] = PR[90,3] + 41.998;
   1:L PR[91] R[100]mm/sec CNT100;
   1:  PR[91,1] = PR[90,1] + -54.130;
   1:  PR[91,2] = PR[90,2] + -18.165;
   1:  PR[91,3] = PR[90,3] + 42.010;
   1:L PR[91] R[100]mm/sec CNT100;
   1:  PR[91,1] = PR[90,1] + -51.553;
   1:  PR[91,2] = PR[90,2] + -16.829;
   1:  PR[91,3] = PR[90,3] + 42.014;
   1:L PR[91] R[100]mm/sec CNT100;
   1:  PR[91,1] = PR[90,1] + -48.667;
   1:  PR[91,2] = PR[90,2] + -14.840;
   1:  PR[91,3] = PR[90,3] + 42.022;
   1:L PR[91] R[100]mm/sec CNT100;
   1:  PR[91,1] = PR[90,1] + -47.858;
   1:  PR[91,2] = PR[90,2] + -14.177;
   1:  PR[91,3] = PR[90,3] + 42.032;
   1:L PR[91] R[100]mm/sec CNT100;
   1:  PR[91,1] = PR[90,1] + -45.179;
   1:  PR[91,2] = PR[90,2] + -11.215;
   1:  PR[91,3] = PR[90,3] + 42.035;
   1:L PR[91] R[100]mm/sec CNT100;
   1:  PR[91,1] = PR[90,1] + -44.479;
   1:  PR[91,2] = PR[90,2] + -10.536;
   1:  PR[91,3] = PR[90,3] + 42.046;
   1:L PR[91] R[100]mm/sec CNT100;
   1:  PR[91,1] = PR[90,1] + -44.176;
   1:  PR[91,2] = PR[90,2] + -10.050;
   1:  PR[91,3] = PR[90,3] + 42.049;
   1:L PR[91] R[100]mm/sec CNT100;
   1:  PR[91,1] = PR[90,1] + -40.501;
   1:  PR[91,2] = PR[90,2] + -3.883;
   1:  PR[91,3] = PR[90,3] + 42.050;
   1:L PR[91] R[100]mm/sec CNT100;
   1:  PR[91,1] = PR[90,1] + -38.678;
   1:  PR[91,2] = PR[90,2] + -8.579;
   1:  PR[91,3] = PR[90,3] + 42.070;
   1:L PR[91] R[100]mm/sec CNT100;
   1:  PR[91,1] = PR[90,1] + -37.842;
   1:  PR[91,2] = PR[90,2] + -10.127;
   1:  PR[91,3] = PR[90,3] + 42.084;
   1:L PR[91] R[100]mm/sec CNT100;
   1:  PR[91,1] = PR[90,1] + -36.990;
   1:  PR[91,2] = PR[90,2] + -11.484;
   1:  PR[91,3] = PR[90,3] + 42.089;
   1:L PR[91] R[100]mm/sec CNT100;
   1:  PR[91,1] = PR[90,1] + -36.742;
   1:  PR[91,2] = PR[90,2] + -11.857;
   1:  PR[91,3] = PR[90,3] + 42.093;
   1:L PR[91] R[100]mm/sec CNT100;
   1:  PR[91,1] = PR[90,1] + -36.258;
   1:  PR[91,2] = PR[90,2] + -12.520;
   1:  PR[91,3] = PR[90,3] + 42.094;
   1:L PR[91] R[100]mm/sec CNT100;
   1:  PR[91,1] = PR[90,1] + -34.502;
   1:  PR[91,2] = PR[90,2] + -14.463;
   1:  PR[91,3] = PR[90,3] + 42.097;
   1:L PR[91] R[100]mm/sec CNT100;
   1:  PR[91,1] = PR[90,1] + -33.197;
   1:  PR[91,2] = PR[90,2] + -15.773;
   1:  PR[91,3] = PR[90,3] + 42.104;
   1:L PR[91] R[100]mm/sec CNT100;
   1:  PR[91,1] = PR[90,1] + -30.812;
   1:  PR[91,2] = PR[90,2] + -17.474;
   1:  PR[91,3] = PR[90,3] + 42.109;
   1:L PR[91] R[100]mm/sec CNT100;
   1:  PR[91,1] = PR[90,1] + -29.551;
   1:  PR[91,2] = PR[90,2] + -18.279;
   1:  PR[91,3] = PR[90,3] + 42.117;
   1:L PR[91] R[100]mm/sec CNT100;
   1:  PR[91,1] = PR[90,1] + -26.411;
   1:  PR[91,2] = PR[90,2] + -19.623;
   1:  PR[91,3] = PR[90,3] + 42.121;
   1:L PR[91] R[100]mm/sec CNT100;
   1:  PR[91,1] = PR[90,1] + -25.429;
   1:  PR[91,2] = PR[90,2] + -19.982;
   1:  PR[91,3] = PR[90,3] + 42.131;
   1:L PR[91] R[100]mm/sec CNT100;
   1:  PR[91,1] = PR[90,1] + -21.515;
   1:  PR[91,2] = PR[90,2] + -20.738;
   1:  PR[91,3] = PR[90,3] + 42.134;
   1:L PR[91] R[100]mm/sec CNT100;
   1:  PR[91,1] = PR[90,1] + -21.015;
   1:  PR[91,2] = PR[90,2] + -20.806;
   1:  PR[91,3] = PR[90,3] + 42.145;
   1:L PR[91] R[100]mm/sec CNT100;
   1:  PR[91,1] = PR[90,1] + -16.444;
   1:  PR[91,2] = PR[90,2] + -20.690;
   1:  PR[91,3] = PR[90,3] + 42.146;
   1:L PR[91] R[100]mm/sec CNT100;
   1:  PR[91,1] = PR[90,1] + -15.743;
   1:  PR[91,2] = PR[90,2] + -20.518;
   1:  PR[91,3] = PR[90,3] + 42.159;
   1:L PR[91] R[100]mm/sec CNT100;
   1:  PR[91,1] = PR[90,1] + -11.846;
   1:  PR[91,2] = PR[90,2] + -19.653;
   1:  PR[91,3] = PR[90,3] + 42.161;
   1:L PR[91] R[100]mm/sec CNT100;
   1:  PR[91,1] = PR[90,1] + -11.425;
   1:  PR[91,2] = PR[90,2] + -19.495;
   1:  PR[91,3] = PR[90,3] + 42.172;
   1:L PR[91] R[100]mm/sec CNT100;
   1:  PR[91,1] = PR[90,1] + -7.622;
   1:  PR[91,2] = PR[90,2] + -17.734;
   1:  PR[91,3] = PR[90,3] + 42.173;
   1:L PR[91] R[100]mm/sec CNT100;
   1:  PR[91,1] = PR[90,1] + -6.581;
   1:  PR[91,2] = PR[90,2] + -17.046;
   1:  PR[91,3] = PR[90,3] + 42.184;
   1:L PR[91] R[100]mm/sec CNT100;
   1:  PR[91,1] = PR[90,1] + -3.877;
   1:  PR[91,2] = PR[90,2] + -14.968;
   1:  PR[91,3] = PR[90,3] + 42.188;
   1:L PR[91] R[100]mm/sec CNT100;
   1:  PR[91,1] = PR[90,1] + -2.525;
   1:  PR[91,2] = PR[90,2] + -13.518;
   1:  PR[91,3] = PR[90,3] + 42.197;
   1:L PR[91] R[100]mm/sec CNT100;
   1:  PR[91,1] = PR[90,1] + -0.835;
   1:  PR[91,2] = PR[90,2] + -11.446;
   1:  PR[91,3] = PR[90,3] + 42.203;
   1:L PR[91] R[100]mm/sec CNT100;
   1:  PR[91,1] = PR[90,1] + 0.280;
   1:  PR[91,2] = PR[90,2] + -9.333;
   1:  PR[91,3] = PR[90,3] + 42.210;
   1:L PR[91] R[100]mm/sec CNT100;
   1:  PR[91,1] = PR[90,1] + 2.362;
   1:  PR[91,2] = PR[90,2] + -4.651;
   1:  PR[91,3] = PR[90,3] + 42.217;
   1:L PR[91] R[100]mm/sec CNT100;
   1:  PR[91,1] = PR[90,1] + 4.247;
   1:  PR[91,2] = PR[90,2] + -9.356;
   1:  PR[91,3] = PR[90,3] + 42.231;
   1:L PR[91] R[100]mm/sec CNT100;
   1:  PR[91,1] = PR[90,1] + 5.341;
   1:  PR[91,2] = PR[90,2] + -11.537;
   1:  PR[91,3] = PR[90,3] + 42.245;
   1:L PR[91] R[100]mm/sec CNT100;
   1:  PR[91,1] = PR[90,1] + 6.684;
   1:  PR[91,2] = PR[90,2] + -13.272;
   1:  PR[91,3] = PR[90,3] + 42.252;
   1:L PR[91] R[100]mm/sec CNT100;
   1:  PR[91,1] = PR[90,1] + 7.497;
   1:  PR[91,2] = PR[90,2] + -14.443;
   1:  PR[91,3] = PR[90,3] + 42.258;
   1:L PR[91] R[100]mm/sec CNT100;
   1:  PR[91,1] = PR[90,1] + 9.240;
   1:  PR[91,2] = PR[90,2] + -16.279;
   1:  PR[91,3] = PR[90,3] + 42.262;
   1:L PR[91] R[100]mm/sec CNT100;
   1:  PR[91,1] = PR[90,1] + 11.590;
   1:  PR[91,2] = PR[90,2] + -18.061;
   1:  PR[91,3] = PR[90,3] + 42.269;
   1:L PR[91] R[100]mm/sec CNT100;
   1:  PR[91,1] = PR[90,1] + 13.626;
   1:  PR[91,2] = PR[90,2] + -19.330;
   1:  PR[91,3] = PR[90,3] + 42.277;
   1:L PR[91] R[100]mm/sec CNT100;
   1:  PR[91,1] = PR[90,1] + 16.503;
   1:  PR[91,2] = PR[90,2] + -20.505;
   1:  PR[91,3] = PR[90,3] + 42.283;
   1:L PR[91] R[100]mm/sec CNT100;
   1:  PR[91,1] = PR[90,1] + 18.636;
   1:  PR[91,2] = PR[90,2] + -21.180;
   1:  PR[91,3] = PR[90,3] + 42.292;
   1:L PR[91] R[100]mm/sec CNT100;
   1:  PR[91,1] = PR[90,1] + 21.888;
   1:  PR[91,2] = PR[90,2] + -21.597;
   1:  PR[91,3] = PR[90,3] + 42.298;
   1:L PR[91] R[100]mm/sec CNT100;
   1:  PR[91,1] = PR[90,1] + 23.948;
   1:  PR[91,2] = PR[90,2] + -21.715;
   1:  PR[91,3] = PR[90,3] + 42.307;
   1:L PR[91] R[100]mm/sec CNT100;
   1:  PR[91,1] = PR[90,1] + 27.367;
   1:  PR[91,2] = PR[90,2] + -21.260;
   1:  PR[91,3] = PR[90,3] + 42.313;
   1:L PR[91] R[100]mm/sec CNT100;
   1:  PR[91,1] = PR[90,1] + 29.223;
   1:  PR[91,2] = PR[90,2] + -20.900;
   1:  PR[91,3] = PR[90,3] + 42.322;
   1:L PR[91] R[100]mm/sec CNT100;
   1:  PR[91,1] = PR[90,1] + 32.558;
   1:  PR[91,2] = PR[90,2] + -19.525;
   1:  PR[91,3] = PR[90,3] + 42.328;
   1:L PR[91] R[100]mm/sec CNT100;
   1:  PR[91,1] = PR[90,1] + 34.123;
   1:  PR[91,2] = PR[90,2] + -18.790;
   1:  PR[91,3] = PR[90,3] + 42.338;
   1:L PR[91] R[100]mm/sec CNT100;
   1:  PR[91,1] = PR[90,1] + 37.251;
   1:  PR[91,2] = PR[90,2] + -16.417;
   1:  PR[91,3] = PR[90,3] + 42.342;
   1:L PR[91] R[100]mm/sec CNT100;
   1:  PR[91,1] = PR[90,1] + 37.451;
   1:  PR[91,2] = PR[90,2] + -16.306;
   1:  PR[91,3] = PR[90,3] + 42.353;
   1:L PR[91] R[100]mm/sec CNT100;
   1:  PR[91,1] = PR[90,1] + 37.538;
   1:  PR[91,2] = PR[90,2] + -16.247;
   1:  PR[91,3] = PR[90,3] + 42.354;
   1:L PR[91] R[100]mm/sec CNT100;
   1:  PR[91,1] = PR[90,1] + 38.587;
   1:  PR[91,2] = PR[90,2] + -15.273;
   1:L PR[91] R[100]mm/sec CNT100;
   1:  PR[91,1] = PR[90,1] + 39.254;
   1:  PR[91,2] = PR[90,2] + -14.542;
   1:  PR[91,3] = PR[90,3] + 42.358;
   1:L PR[91] R[100]mm/sec CNT100;
   1:  PR[91,1] = PR[90,1] + 40.916;
   1:  PR[91,2] = PR[90,2] + -12.537;
   1:  PR[91,3] = PR[90,3] + 42.361;
   1:L PR[91] R[100]mm/sec CNT100;
   1:  PR[91,1] = PR[90,1] + 42.629;
   1:  PR[91,2] = PR[90,2] + -14.275;
   1:  PR[91,3] = PR[90,3] + 42.368;
   1:L PR[91] R[100]mm/sec CNT100;
   1:  PR[91,1] = PR[90,1] + 45.919;
   1:  PR[91,2] = PR[90,2] + -16.624;
   1:  PR[91,3] = PR[90,3] + 42.375;
   1:L PR[91] R[100]mm/sec CNT100;
   1:  PR[91,1] = PR[90,1] + 48.337;
   1:  PR[91,2] = PR[90,2] + -18.206;
   1:  PR[91,3] = PR[90,3] + 42.386;
   1:L PR[91] R[100]mm/sec CNT100;
   1:  PR[91,1] = PR[90,1] + 49.626;
   1:  PR[91,2] = PR[90,2] + -18.748;
   1:  PR[91,3] = PR[90,3] + 42.394;
   1:L PR[91] R[100]mm/sec CNT100;
   1:  PR[91,1] = PR[90,1] + 52.266;
   1:  PR[91,2] = PR[90,2] + -19.767;
   1:  PR[91,3] = PR[90,3] + 42.398;
   1:L PR[91] R[100]mm/sec CNT100;
   1:  PR[91,1] = PR[90,1] + 54.093;
   1:  PR[91,2] = PR[90,2] + -20.565;
   1:  PR[91,3] = PR[90,3] + 42.406;
   1:L PR[91] R[100]mm/sec CNT100;
   1:  PR[91,1] = PR[90,1] + 54.942;
   1:  PR[91,2] = PR[90,2] + -20.851;
   1:  PR[91,3] = PR[90,3] + 42.411;
   1:L PR[91] R[100]mm/sec CNT100;
   1:  PR[91,1] = PR[90,1] + 58.727;
   1:  PR[91,2] = PR[90,2] + -21.656;
   1:  PR[91,3] = PR[90,3] + 42.414;
   1:L PR[91] R[100]mm/sec CNT100;
   1:  PR[91,1] = PR[90,1] + 62.409;
   1:  PR[91,2] = PR[90,2] + -22.070;
   1:  PR[91,3] = PR[90,3] + 42.424;
   1:L PR[91] R[100]mm/sec CNT100;
   1:  PR[91,1] = PR[90,1] + 63.754;
   1:  PR[91,2] = PR[90,2] + -22.094;
   1:  PR[91,3] = PR[90,3] + 42.434;
   1:L PR[91] R[100]mm/sec CNT100;
   1:  PR[91,1] = PR[90,1] + 67.262;
   1:  PR[91,2] = PR[90,2] + -21.775;
   1:  PR[91,3] = PR[90,3] + 42.438;
   1:L PR[91] R[100]mm/sec CNT100;
   1:  PR[91,1] = PR[90,1] + 69.083;
   1:  PR[91,2] = PR[90,2] + -21.648;
   1:  PR[91,3] = PR[90,3] + 42.448;
   1:L PR[91] R[100]mm/sec CNT100;
   1:  PR[91,1] = PR[90,1] + 69.444;
   1:  PR[91,2] = PR[90,2] + -21.588;
   1:  PR[91,3] = PR[90,3] + 42.453;
   1:L PR[91] R[100]mm/sec CNT100;
   1:  PR[91,1] = PR[90,1] + 73.643;
   1:  PR[91,2] = PR[90,2] + -20.355;
   1:  PR[91,3] = PR[90,3] + 42.454;
   1:L PR[91] R[100]mm/sec CNT100;
   1:  PR[91,1] = PR[90,1] + 75.212;
   1:  PR[91,2] = PR[90,2] + -19.754;
   1:  PR[91,3] = PR[90,3] + 42.466;
   1:L PR[91] R[100]mm/sec CNT100;
   1:  PR[91,1] = PR[90,1] + 77.743;
   1:  PR[91,2] = PR[90,2] + -18.356;
   1:  PR[91,3] = PR[90,3] + 42.471;
   1:L PR[91] R[100]mm/sec CNT100;
   1:  PR[91,1] = PR[90,1] + 79.954;
   1:  PR[91,2] = PR[90,2] + -16.939;
   1:  PR[91,3] = PR[90,3] + 42.479;
   1:L PR[91] R[100]mm/sec CNT100;
   1:  PR[91,1] = PR[90,1] + 81.304;
   1:  PR[91,2] = PR[90,2] + -15.734;
   1:  PR[91,3] = PR[90,3] + 42.486;
   1:L PR[91] R[100]mm/sec CNT100;
   1:  PR[91,1] = PR[90,1] + 83.634;
   1:  PR[91,2] = PR[90,2] + -13.427;
   1:  PR[91,3] = PR[90,3] + 42.491;
   1:L PR[91] R[100]mm/sec CNT100;
   1:  PR[91,1] = PR[90,1] + 84.235;
   1:  PR[91,2] = PR[90,2] + -12.565;
   1:  PR[91,3] = PR[90,3] + 42.500;
   1:L PR[91] R[100]mm/sec CNT100;
   1:  PR[91,1] = PR[90,1] + 86.250;
   1:  PR[91,2] = PR[90,2] + -9.439;
   1:  PR[91,3] = PR[90,3] + 42.503;
   1:L PR[91] R[100]mm/sec CNT100;
   1:  PR[91,1] = PR[90,1] + 86.449;
   1:  PR[91,2] = PR[90,2] + -8.925;
   1:  PR[91,3] = PR[90,3] + 42.513;
   1:L PR[91] R[100]mm/sec CNT100;
   1:  PR[91,1] = PR[90,1] + 87.810;
   1:  PR[91,2] = PR[90,2] + -5.162;
   1:  PR[91,3] = PR[90,3] + 42.515;
   1:L PR[91] R[100]mm/sec CNT100;
   1:  PR[91,1] = PR[90,1] + 88.326;
   1:  PR[91,2] = PR[90,2] + -0.792;
   1:  PR[91,3] = PR[90,3] + 42.526;
   1:L PR[91] R[100]mm/sec CNT100;
   1:  PR[91,1] = PR[90,1] + 88.363;
   1:  PR[91,2] = PR[90,2] + -0.627;
   1:  PR[91,3] = PR[90,3] + 42.538;
   1:L PR[91] R[100]mm/sec CNT100;
   1:  PR[91,1] = PR[90,1] + 88.229;
   1:  PR[91,2] = PR[90,2] + 0.528;
   1:L PR[91] R[100]mm/sec CNT100;
   1:  PR[91,1] = PR[90,1] + 87.815;
   1:  PR[91,2] = PR[90,2] + 3.691;
   1:  PR[91,3] = PR[90,3] + 42.541;
   1:L PR[91] R[100]mm/sec CNT100;
   1:  PR[91,1] = PR[90,1] + 86.449;
   1:  PR[91,2] = PR[90,2] + 7.466;
   1:  PR[91,3] = PR[90,3] + 42.550;
   1:L PR[91] R[100]mm/sec CNT100;
   1:  PR[91,1] = PR[90,1] + 86.251;
   1:  PR[91,2] = PR[90,2] + 7.980;
   1:  PR[91,3] = PR[90,3] + 42.561;
   1:L PR[91] R[100]mm/sec CNT100;
   1:  PR[91,1] = PR[90,1] + 84.235;
   1:  PR[91,2] = PR[90,2] + 11.106;
   1:  PR[91,3] = PR[90,3] + 42.563;
   1:L PR[91] R[100]mm/sec CNT100;
   1:  PR[91,1] = PR[90,1] + 83.634;
   1:  PR[91,2] = PR[90,2] + 11.968;
   1:  PR[91,3] = PR[90,3] + 42.573;
   1:L PR[91] R[100]mm/sec CNT100;
   1:  PR[91,1] = PR[90,1] + 81.304;
   1:  PR[91,2] = PR[90,2] + 14.275;
   1:  PR[91,3] = PR[90,3] + 42.576;
   1:L PR[91] R[100]mm/sec CNT100;
   1:  PR[91,1] = PR[90,1] + 79.954;
   1:  PR[91,2] = PR[90,2] + 15.480;
   1:  PR[91,3] = PR[90,3] + 42.585;
   1:L PR[91] R[100]mm/sec CNT100;
   1:  PR[91,1] = PR[90,1] + 77.744;
   1:  PR[91,2] = PR[90,2] + 16.897;
   1:  PR[91,3] = PR[90,3] + 42.590;
   1:L PR[91] R[100]mm/sec CNT100;
   1:  PR[91,1] = PR[90,1] + 75.213;
   1:  PR[91,2] = PR[90,2] + 18.295;
   1:  PR[91,3] = PR[90,3] + 42.597;
   1:L PR[91] R[100]mm/sec CNT100;
   1:  PR[91,1] = PR[90,1] + 73.643;
   1:  PR[91,2] = PR[90,2] + 18.896;
   1:  PR[91,3] = PR[90,3] + 42.605;
   1:L PR[91] R[100]mm/sec CNT100;
   1:  PR[91,1] = PR[90,1] + 69.445;
   1:  PR[91,2] = PR[90,2] + 20.129;
   1:  PR[91,3] = PR[90,3] + 42.610;
   1:L PR[91] R[100]mm/sec CNT100;
   1:  PR[91,1] = PR[90,1] + 69.084;
   1:  PR[91,2] = PR[90,2] + 20.189;
   1:  PR[91,3] = PR[90,3] + 42.622;
   1:L PR[91] R[100]mm/sec CNT100;
   1:  PR[91,1] = PR[90,1] + 67.262;
   1:  PR[91,2] = PR[90,2] + 20.316;
   1:  PR[91,3] = PR[90,3] + 42.623;
   1:L PR[91] R[100]mm/sec CNT100;
   1:  PR[91,1] = PR[90,1] + 63.746;
   1:  PR[91,2] = PR[90,2] + 20.636;
   1:  PR[91,3] = PR[90,3] + 42.628;
   1:L PR[91] R[100]mm/sec CNT100;
   1:  PR[91,1] = PR[90,1] + 62.381;
   1:  PR[91,2] = PR[90,2] + 20.609;
   1:  PR[91,3] = PR[90,3] + 42.638;
   1:L PR[91] R[100]mm/sec CNT100;
   1:  PR[91,1] = PR[90,1] + 58.696;
   1:  PR[91,2] = PR[90,2] + 20.194;
   1:  PR[91,3] = PR[90,3] + 42.642;
   1:L PR[91] R[100]mm/sec CNT100;
   1:  PR[91,1] = PR[90,1] + 54.857;
   1:  PR[91,2] = PR[90,2] + 19.366;
   1:  PR[91,3] = PR[90,3] + 42.652;
   1:L PR[91] R[100]mm/sec CNT100;
   1:  PR[91,1] = PR[90,1] + 54.036;
   1:  PR[91,2] = PR[90,2] + 19.090;
   1:  PR[91,3] = PR[90,3] + 42.663;
   1:L PR[91] R[100]mm/sec CNT100;
   1:  PR[91,1] = PR[90,1] + 52.273;
   1:  PR[91,2] = PR[90,2] + 18.312;
   1:  PR[91,3] = PR[90,3] + 42.665;
   1:L PR[91] R[100]mm/sec CNT100;
   1:  PR[91,1] = PR[90,1] + 49.579;
   1:  PR[91,2] = PR[90,2] + 17.261;
   1:  PR[91,3] = PR[90,3] + 42.670;
   1:L PR[91] R[100]mm/sec CNT100;
   1:  PR[91,1] = PR[90,1] + 48.285;
   1:  PR[91,2] = PR[90,2] + 16.721;
   1:  PR[91,3] = PR[90,3] + 42.678;
   1:L PR[91] R[100]mm/sec CNT100;
   1:  PR[91,1] = PR[90,1] + 45.909;
   1:  PR[91,2] = PR[90,2] + 15.149;
   1:  PR[91,3] = PR[90,3] + 42.682;
   1:L PR[91] R[100]mm/sec CNT100;
   1:  PR[91,1] = PR[90,1] + 42.647;
   1:  PR[91,2] = PR[90,2] + 12.830;
   1:  PR[91,3] = PR[90,3] + 42.690;
   1:L PR[91] R[100]mm/sec CNT100;
   1:  PR[91,1] = PR[90,1] + 40.899;
   1:  PR[91,2] = PR[90,2] + 10.980;
   1:  PR[91,3] = PR[90,3] + 42.701;
   1:L PR[91] R[100]mm/sec CNT100;
   1:  PR[91,1] = PR[90,1] + 39.253;
   1:  PR[91,2] = PR[90,2] + 13.080;
   1:  PR[91,3] = PR[90,3] + 42.708;
   1:L PR[91] R[100]mm/sec CNT100;
   1:  PR[91,1] = PR[90,1] + 37.453;
   1:  PR[91,2] = PR[90,2] + 14.864;
   1:  PR[91,3] = PR[90,3] + 42.716;
   1:L PR[91] R[100]mm/sec CNT100;
   1:  PR[91,1] = PR[90,1] + 34.921;
   1:  PR[91,2] = PR[90,2] + 16.779;
   1:  PR[91,3] = PR[90,3] + 42.723;
   1:L PR[91] R[100]mm/sec CNT100;
   1:  PR[91,1] = PR[90,1] + 34.339;
   1:  PR[91,2] = PR[90,2] + 17.198;
   1:  PR[91,3] = PR[90,3] + 42.731;
   1:L PR[91] R[100]mm/sec CNT100;
   1:  PR[91,1] = PR[90,1] + 34.156;
   1:  PR[91,2] = PR[90,2] + 17.319;
   1:  PR[91,3] = PR[90,3] + 42.733;
   1:L PR[91] R[100]mm/sec CNT100;
   1:  PR[91,1] = PR[90,1] + 32.533;
   1:  PR[91,2] = PR[90,2] + 18.081;
   1:  PR[91,3] = PR[90,3] + 42.734;
   1:L PR[91] R[100]mm/sec CNT100;
   1:  PR[91,1] = PR[90,1] + 29.200;
   1:  PR[91,2] = PR[90,2] + 19.448;
   1:  PR[91,3] = PR[90,3] + 42.739;
   1:L PR[91] R[100]mm/sec CNT100;
   1:  PR[91,1] = PR[90,1] + 27.344;
   1:  PR[91,2] = PR[90,2] + 19.807;
   1:  PR[91,3] = PR[90,3] + 42.749;
   1:L PR[91] R[100]mm/sec CNT100;
   1:  PR[91,1] = PR[90,1] + 23.929;
   1:  PR[91,2] = PR[90,2] + 20.256;
   1:  PR[91,3] = PR[90,3] + 42.754;
   1:L PR[91] R[100]mm/sec CNT100;
   1:  PR[91,1] = PR[90,1] + 21.870;
   1:  PR[91,2] = PR[90,2] + 20.138;
   1:  PR[91,3] = PR[90,3] + 42.764;
   1:L PR[91] R[100]mm/sec CNT100;
   1:  PR[91,1] = PR[90,1] + 18.623;
   1:  PR[91,2] = PR[90,2] + 19.718;
   1:  PR[91,3] = PR[90,3] + 42.769;
   1:L PR[91] R[100]mm/sec CNT100;
   1:  PR[91,1] = PR[90,1] + 16.491;
   1:  PR[91,2] = PR[90,2] + 19.044;
   1:  PR[91,3] = PR[90,3] + 42.778;
   1:L PR[91] R[100]mm/sec CNT100;
   1:  PR[91,1] = PR[90,1] + 13.619;
   1:  PR[91,2] = PR[90,2] + 17.867;
   1:  PR[91,3] = PR[90,3] + 42.784;
   1:L PR[91] R[100]mm/sec CNT100;
   1:  PR[91,1] = PR[90,1] + 11.583;
   1:  PR[91,2] = PR[90,2] + 16.600;
   1:  PR[91,3] = PR[90,3] + 42.793;
   1:L PR[91] R[100]mm/sec CNT100;
   1:  PR[91,1] = PR[90,1] + 9.238;
   1:  PR[91,2] = PR[90,2] + 14.818;
   1:  PR[91,3] = PR[90,3] + 42.800;
   1:L PR[91] R[100]mm/sec CNT100;
   1:  PR[91,1] = PR[90,1] + 7.460;
   1:  PR[91,2] = PR[90,2] + 12.947;
   1:  PR[91,3] = PR[90,3] + 42.808;
   1:L PR[91] R[100]mm/sec CNT100;
   1:  PR[91,1] = PR[90,1] + 5.718;
   1:  PR[91,2] = PR[90,2] + 10.696;
   1:  PR[91,3] = PR[90,3] + 42.815;
   1:L PR[91] R[100]mm/sec CNT100;
   1:  PR[91,1] = PR[90,1] + 5.478;
   1:  PR[91,2] = PR[90,2] + 10.324;
   1:  PR[91,3] = PR[90,3] + 42.823;
   1:L PR[91] R[100]mm/sec CNT100;
   1:  PR[91,1] = PR[90,1] + 4.531;
   1:  PR[91,2] = PR[90,2] + 8.514;
   1:  PR[91,3] = PR[90,3] + 42.824;
   1:L PR[91] R[100]mm/sec CNT100;
   1:  PR[91,1] = PR[90,1] + 2.356;
   1:  PR[91,2] = PR[90,2] + 3.204;
   1:  PR[91,3] = PR[90,3] + 42.830;
   1:L PR[91] R[100]mm/sec CNT100;
   1:  PR[91,1] = PR[90,1] + -0.033;
   1:  PR[91,2] = PR[90,2] + 8.509;
   1:  PR[91,3] = PR[90,3] + 42.845;
   1:L PR[91] R[100]mm/sec CNT100;
   1:  PR[91,1] = PR[90,1] + -0.817;
   1:  PR[91,2] = PR[90,2] + 9.961;
   1:  PR[91,3] = PR[90,3] + 42.862;
   1:L PR[91] R[100]mm/sec CNT100;
   1:  PR[91,1] = PR[90,1] + -2.504;
   1:  PR[91,2] = PR[90,2] + 12.033;
   1:  PR[91,3] = PR[90,3] + 42.866;
   1:L PR[91] R[100]mm/sec CNT100;
   1:  PR[91,1] = PR[90,1] + -3.863;
   1:  PR[91,2] = PR[90,2] + 13.496;
   1:  PR[91,3] = PR[90,3] + 42.873;
   1:L PR[91] R[100]mm/sec CNT100;
   1:  PR[91,1] = PR[90,1] + -6.563;
   1:  PR[91,2] = PR[90,2] + 15.574;
   1:  PR[91,3] = PR[90,3] + 42.879;
   1:L PR[91] R[100]mm/sec CNT100;
   1:  PR[91,1] = PR[90,1] + -7.606;
   1:  PR[91,2] = PR[90,2] + 16.266;
   1:  PR[91,3] = PR[90,3] + 42.888;
   1:L PR[91] R[100]mm/sec CNT100;
   1:  PR[91,1] = PR[90,1] + -11.407;
   1:  PR[91,2] = PR[90,2] + 18.029;
   1:  PR[91,3] = PR[90,3] + 42.892;
   1:L PR[91] R[100]mm/sec CNT100;
   1:  PR[91,1] = PR[90,1] + -11.831;
   1:  PR[91,2] = PR[90,2] + 18.189;
   1:  PR[91,3] = PR[90,3] + 42.903;
   1:L PR[91] R[100]mm/sec CNT100;
   1:  PR[91,1] = PR[90,1] + -15.744;
   1:  PR[91,2] = PR[90,2] + 19.061;
   1:  PR[91,3] = PR[90,3] + 42.905;
   1:L PR[91] R[100]mm/sec CNT100;
   1:  PR[91,1] = PR[90,1] + -16.430;
   1:  PR[91,2] = PR[90,2] + 19.229;
   1:  PR[91,3] = PR[90,3] + 42.916;
   1:L PR[91] R[100]mm/sec CNT100;
   1:  PR[91,1] = PR[90,1] + -21.003;
   1:  PR[91,2] = PR[90,2] + 19.348;
   1:  PR[91,3] = PR[90,3] + 42.918;
   1:L PR[91] R[100]mm/sec CNT100;
   1:  PR[91,1] = PR[90,1] + -21.502;
   1:  PR[91,2] = PR[90,2] + 19.280;
   1:  PR[91,3] = PR[90,3] + 42.930;
   1:L PR[91] R[100]mm/sec CNT100;
   1:  PR[91,1] = PR[90,1] + -25.419;
   1:  PR[91,2] = PR[90,2] + 18.526;
   1:  PR[91,3] = PR[90,3] + 42.932;
   1:L PR[91] R[100]mm/sec CNT100;
   1:  PR[91,1] = PR[90,1] + -26.400;
   1:  PR[91,2] = PR[90,2] + 18.167;
   1:  PR[91,3] = PR[90,3] + 42.943;
   1:L PR[91] R[100]mm/sec CNT100;
   1:  PR[91,1] = PR[90,1] + -29.543;
   1:  PR[91,2] = PR[90,2] + 16.824;
   1:  PR[91,3] = PR[90,3] + 42.946;
   1:L PR[91] R[100]mm/sec CNT100;
   1:  PR[91,1] = PR[90,1] + -30.804;
   1:  PR[91,2] = PR[90,2] + 16.020;
   1:  PR[91,3] = PR[90,3] + 42.955;
   1:L PR[91] R[100]mm/sec CNT100;
   1:  PR[91,1] = PR[90,1] + -33.192;
   1:  PR[91,2] = PR[90,2] + 14.319;
   1:  PR[91,3] = PR[90,3] + 42.959;
   1:L PR[91] R[100]mm/sec CNT100;
   1:  PR[91,1] = PR[90,1] + -34.496;
   1:  PR[91,2] = PR[90,2] + 13.010;
   1:  PR[91,3] = PR[90,3] + 42.967;
   1:L PR[91] R[100]mm/sec CNT100;
   1:  PR[91,1] = PR[90,1] + -36.206;
   1:  PR[91,2] = PR[90,2] + 11.119;
   1:  PR[91,3] = PR[90,3] + 42.972;
   1:L PR[91] R[100]mm/sec CNT100;
   1:  PR[91,1] = PR[90,1] + -37.416;
   1:  PR[91,2] = PR[90,2] + 9.200;
   1:  PR[91,3] = PR[90,3] + 42.979;
   1:L PR[91] R[100]mm/sec CNT100;
   1:  PR[91,1] = PR[90,1] + -37.697;
   1:  PR[91,2] = PR[90,2] + 8.858;
   1:  PR[91,3] = PR[90,3] + 42.986;
   1:L PR[91] R[100]mm/sec CNT100;
   1:  PR[91,1] = PR[90,1] + -38.132;
   1:  PR[91,2] = PR[90,2] + 8.196;
   1:  PR[91,3] = PR[90,3] + 42.987;
   1:L PR[91] R[100]mm/sec CNT100;
   1:  PR[91,1] = PR[90,1] + -38.601;
   1:  PR[91,2] = PR[90,2] + 7.287;
   1:  PR[91,3] = PR[90,3] + 42.989;
   1:L PR[91] R[100]mm/sec CNT100;
   1:  PR[91,1] = PR[90,1] + -38.838;
   1:  PR[91,2] = PR[90,2] + 6.608;
   1:  PR[91,3] = PR[90,3] + 42.992;
   1:L PR[91] R[100]mm/sec CNT100;
   1:  PR[91,1] = PR[90,1] + -38.983;
   1:  PR[91,2] = PR[90,2] + 6.371;
   1:  PR[91,3] = PR[90,3] + 42.994;
   1:L PR[91] R[100]mm/sec CNT100;
   1:  PR[91,1] = PR[90,1] + -40.785;
   1:  PR[91,2] = PR[90,2] + 1.866;
   1:  PR[91,3] = PR[90,3] + 42.995;
   1:L PR[91] R[100]mm/sec CNT100;
   1:  PR[91,1] = PR[90,1] + -43.156;
   1:  PR[91,2] = PR[90,2] + 7.175;
   1:  PR[91,3] = PR[90,3] + 43.008;
   1:L PR[91] R[100]mm/sec CNT100;
   1:  PR[91,1] = PR[90,1] + -45.002;
   1:  PR[91,2] = PR[90,2] + 9.708;
   1:  PR[91,3] = PR[90,3] + 43.024;
   1:L PR[91] R[100]mm/sec CNT100;
   1:  PR[91,1] = PR[90,1] + -46.307;
   1:  PR[91,2] = PR[90,2] + 11.307;
   1:  PR[91,3] = PR[90,3] + 43.033;
   1:L PR[91] R[100]mm/sec CNT100;
   1:  PR[91,1] = PR[90,1] + -47.680;
   1:  PR[91,2] = PR[90,2] + 12.468;
   1:  PR[91,3] = PR[90,3] + 43.038;
   1:L PR[91] R[100]mm/sec CNT100;
   1:  PR[91,1] = PR[90,1] + -50.578;
   1:  PR[91,2] = PR[90,2] + 14.710;
   1:  PR[91,3] = PR[90,3] + 43.043;
   1:L PR[91] R[100]mm/sec CNT100;
   1:  PR[91,1] = PR[90,1] + -51.638;
   1:  PR[91,2] = PR[90,2] + 15.241;
   1:  PR[91,3] = PR[90,3] + 43.054;
   1:L PR[91] R[100]mm/sec CNT100;
   1:  PR[91,1] = PR[90,1] + -55.124;
   1:  PR[91,2] = PR[90,2] + 17.139;
   1:  PR[91,3] = PR[90,3] + 43.057;
   1:L PR[91] R[100]mm/sec CNT100;
   1:  PR[91,1] = PR[90,1] + -56.657;
   1:  PR[91,2] = PR[90,2] + 17.635;
   1:  PR[91,3] = PR[90,3] + 43.068;
   1:L PR[91] R[100]mm/sec CNT100;
   1:  PR[91,1] = PR[90,1] + -59.822;
   1:  PR[91,2] = PR[90,2] + 18.626;
   1:  PR[91,3] = PR[90,3] + 43.072;
   1:L PR[91] R[100]mm/sec CNT100;
   1:  PR[91,1] = PR[90,1] + -64.715;
   1:  PR[91,2] = PR[90,2] + 19.237;
   1:  PR[91,3] = PR[90,3] + 43.081;
   1:L PR[91] R[100]mm/sec CNT100;
   1:  PR[91] = PR[90];
   1:  PR[91,1] = PR[90,1] + -68.880;
   1:  PR[91,2] = PR[90,2] + 19.120;
   1:  PR[91,3] = PR[90,3] + 44.395;
   1:L PR[91] R[100]mm/sec CNT100;
   1:  PR[91,1] = PR[90,1] + -73.343;
   1:  PR[91,2] = PR[90,2] + 18.041;
   1:  PR[91,3] = PR[90,3] + 43.109;
   1:L PR[91] R[100]mm/sec CNT100;
   1:  PR[91,1] = PR[90,1] + -77.371;
   1:  PR[91,2] = PR[90,2] + 16.200;
   1:  PR[91,3] = PR[90,3] + 43.122;
   1:L PR[91] R[100]mm/sec CNT100;
   1:  PR[91,1] = PR[90,1] + -80.882;
   1:  PR[91,2] = PR[90,2] + 13.676;
   1:  PR[91,3] = PR[90,3] + 43.135;
   1:L PR[91] R[100]mm/sec CNT100;
   1:  PR[91,1] = PR[90,1] + -82.433;
   1:  PR[91,2] = PR[90,2] + 12.009;
   1:  PR[91,3] = PR[90,3] + 43.147;
   1:L PR[91] R[100]mm/sec CNT100;
   1:  PR[91,1] = PR[90,1] + -83.736;
   1:  PR[91,2] = PR[90,2] + 10.591;
   1:  PR[91,3] = PR[90,3] + 43.154;
   1:L PR[91] R[100]mm/sec CNT100;
   1:  PR[91,1] = PR[90,1] + -85.850;
   1:  PR[91,2] = PR[90,2] + 7.062;
   1:  PR[91,3] = PR[90,3] + 43.159;
   1:L PR[91] R[100]mm/sec CNT100;
   1:  PR[91,1] = PR[90,1] + -87.144;
   1:  PR[91,2] = PR[90,2] + 3.240;
   1:  PR[91,3] = PR[90,3] + 43.171;
   1:L PR[91] R[100]mm/sec CNT100;
   1:  PR[91,1] = PR[90,1] + -87.486;
   1:  PR[91,2] = PR[90,2] + 0.145;
   1:  PR[91,3] = PR[90,3] + 43.182;
   1:L PR[91] R[100]mm/sec CNT100;
   1:  PR[91,1] = PR[90,1] + -87.649;
   1:  PR[91,2] = PR[90,2] + -0.688;
   1:  PR[91,3] = PR[90,3] + 43.191;
   1:L PR[91] R[100]mm/sec CNT100;
   1:  PR[91,1] = PR[90,1] + -87.647;
   1:  PR[91,2] = PR[90,2] + -0.699;
   1:  PR[91,3] = PR[90,3] + 43.194;
   1:L PR[91] R[100]mm/sec CNT100;
   1:  PR[91,1] = PR[90,1] + -87.219;
   1:  PR[91,2] = PR[90,2] + -4.708;
   1:L PR[91] R[100]mm/sec CNT100;
   1:  PR[91,1] = PR[90,1] + -85.958;
   1:  PR[91,2] = PR[90,2] + -8.531;
   1:  PR[91,3] = PR[90,3] + 43.205;
   1:L PR[91] R[100]mm/sec CNT100;
   1:  PR[91,1] = PR[90,1] + -85.558;
   1:  PR[91,2] = PR[90,2] + -9.215;
   1:  PR[91,3] = PR[90,3] + 43.217;
   1:L PR[91] R[100]mm/sec CNT100;
   1:  PR[91,1] = PR[90,1] + -83.846;
   1:  PR[91,2] = PR[90,2] + -12.026;
   1:  PR[91,3] = PR[90,3] + 43.219;
   1:L PR[91] R[100]mm/sec CNT100;
   1:  PR[91,1] = PR[90,1] + -80.941;
   1:  PR[91,2] = PR[90,2] + -15.119;
   1:  PR[91,3] = PR[90,3] + 43.229;
   1:L PR[91] R[100]mm/sec CNT100;
   1:  PR[91,1] = PR[90,1] + -78.191;
   1:  PR[91,2] = PR[90,2] + -17.056;
   1:  PR[91,3] = PR[90,3] + 43.241;
   1:L PR[91] R[100]mm/sec CNT100;
   1:  PR[91,1] = PR[90,1] + -77.361;
   1:  PR[91,2] = PR[90,2] + -17.655;
   1:  PR[91,3] = PR[90,3] + 43.250;
   1:L PR[91] R[100]mm/sec CNT100;
   1:  PR[91,1] = PR[90,1] + -74.804;
   1:  PR[91,2] = PR[90,2] + -18.794;
   1:  PR[91,3] = PR[90,3] + 43.253;
   1:L PR[91] R[100]mm/sec CNT100;
   1:  PR[91,1] = PR[90,1] + -73.253;
   1:  PR[91,2] = PR[90,2] + -19.510;
   1:  PR[91,3] = PR[90,3] + 43.261;
   1:L PR[91] R[100]mm/sec CNT100;
   1:  PR[91,1] = PR[90,1] + -71.208;
   1:  PR[91,2] = PR[90,2] + -19.986;
   1:  PR[91,3] = PR[90,3] + 43.266;
   1:L PR[91] R[100]mm/sec CNT100;
   1:  PR[91,1] = PR[90,1] + -68.761;
   1:  PR[91,2] = PR[90,2] + -20.595;
   1:  PR[91,3] = PR[90,3] + 43.272;
   1:L PR[91] R[100]mm/sec CNT100;
   1:  PR[91,1] = PR[90,1] + -67.502;
   1:  PR[91,2] = PR[90,2] + -20.646;
   1:  PR[91,3] = PR[90,3] + 43.279;
   1:L PR[91] R[100]mm/sec CNT100;
   1:  PR[91,1] = PR[90,1] + -64.046;
   1:  PR[91,2] = PR[90,2] + -20.845;
   1:  PR[91,3] = PR[90,3] + 43.283;
   1:L PR[91] R[100]mm/sec CNT100;
   1:  PR[91,1] = PR[90,1] + -61.882;
   1:  PR[91,2] = PR[90,2] + -20.554;
   1:  PR[91,3] = PR[90,3] + 43.293;
   1:L PR[91] R[100]mm/sec CNT100;
   1:  PR[91,1] = PR[90,1] + -59.377;
   1:  PR[91,2] = PR[90,2] + -20.283;
   1:  PR[91,3] = PR[90,3] + 43.299;
   1:L PR[91] R[100]mm/sec CNT100;
   1:  PR[91,1] = PR[90,1] + -58.592;
   1:  PR[91,2] = PR[90,2] + -20.127;
   1:  PR[91,3] = PR[90,3] + 43.306;
   1:L PR[91] R[100]mm/sec CNT100;
   1:  PR[91,1] = PR[90,1] + -55.081;
   1:  PR[91,2] = PR[90,2] + -19.088;
   1:  PR[91,3] = PR[90,3] + 43.309;
   1:L PR[91] R[100]mm/sec CNT100;
   1:  PR[91,1] = PR[90,1] + -52.515;
   1:  PR[91,2] = PR[90,2] + -18.026;
   1:  PR[91,3] = PR[90,3] + 43.319;
   1:L PR[91] R[100]mm/sec CNT100;
   1:  PR[91,1] = PR[90,1] + -50.939;
   1:  PR[91,2] = PR[90,2] + -17.209;
   1:  PR[91,3] = PR[90,3] + 43.327;
   1:L PR[91] R[100]mm/sec CNT100;
   1:  PR[91,1] = PR[90,1] + -47.055;
   1:  PR[91,2] = PR[90,2] + -14.525;
   1:  PR[91,3] = PR[90,3] + 43.332;
   1:L PR[91] R[100]mm/sec CNT100;
   1:  PR[91,1] = PR[90,1] + -47.017;
   1:  PR[91,2] = PR[90,2] + -14.482;
   1:  PR[91,3] = PR[90,3] + 43.345;
   1:L PR[91] R[100]mm/sec CNT100;
   1:  PR[91,1] = PR[90,1] + -43.138;
   1:  PR[91,2] = PR[90,2] + -10.722;
   1:  PR[91,3] = PR[90,3] + 43.346;
   1:L PR[91] R[100]mm/sec CNT100;
   1:  PR[91,1] = PR[90,1] + -40.020;
   1:  PR[91,2] = PR[90,2] + -5.739;
   1:  PR[91,3] = PR[90,3] + 43.361;
   1:L PR[91] R[100]mm/sec CNT100;
   1:  PR[91,1] = PR[90,1] + -37.515;
   1:  PR[91,2] = PR[90,2] + -10.380;
   1:  PR[91,3] = PR[90,3] + 43.378;
   1:L PR[91] R[100]mm/sec CNT100;
   1:  PR[91,1] = PR[90,1] + -36.963;
   1:  PR[91,2] = PR[90,2] + -11.258;
   1:  PR[91,3] = PR[90,3] + 43.393;
   1:L PR[91] R[100]mm/sec CNT100;
   1:  PR[91,1] = PR[90,1] + -36.662;
   1:  PR[91,2] = PR[90,2] + -11.709;
   1:  PR[91,3] = PR[90,3] + 43.396;
   1:L PR[91] R[100]mm/sec CNT100;
   1:  PR[91,1] = PR[90,1] + -36.076;
   1:  PR[91,2] = PR[90,2] + -12.513;
   1:  PR[91,3] = PR[90,3] + 43.397;
   1:L PR[91] R[100]mm/sec CNT100;
   1:  PR[91,1] = PR[90,1] + -33.984;
   1:  PR[91,2] = PR[90,2] + -14.829;
   1:  PR[91,3] = PR[90,3] + 43.400;
   1:L PR[91] R[100]mm/sec CNT100;
   1:  PR[91,1] = PR[90,1] + -33.019;
   1:  PR[91,2] = PR[90,2] + -15.797;
   1:  PR[91,3] = PR[90,3] + 43.409;
   1:L PR[91] R[100]mm/sec CNT100;
   1:  PR[91,1] = PR[90,1] + -30.208;
   1:  PR[91,2] = PR[90,2] + -17.801;
   1:  PR[91,3] = PR[90,3] + 43.413;
   1:L PR[91] R[100]mm/sec CNT100;
   1:  PR[91,1] = PR[90,1] + -29.372;
   1:  PR[91,2] = PR[90,2] + -18.335;
   1:  PR[91,3] = PR[90,3] + 43.423;
   1:L PR[91] R[100]mm/sec CNT100;
   1:  PR[91,1] = PR[90,1] + -25.729;
   1:  PR[91,2] = PR[90,2] + -19.895;
   1:  PR[91,3] = PR[90,3] + 43.426;
   1:L PR[91] R[100]mm/sec CNT100;
   1:  PR[91,1] = PR[90,1] + -25.244;
   1:  PR[91,2] = PR[90,2] + -20.072;
   1:  PR[91,3] = PR[90,3] + 43.437;
   1:L PR[91] R[100]mm/sec CNT100;
   1:  PR[91,1] = PR[90,1] + -20.801;
   1:  PR[91,2] = PR[90,2] + -20.930;
   1:  PR[91,3] = PR[90,3] + 43.439;
   1:L PR[91] R[100]mm/sec CNT100;
   1:  PR[91,1] = PR[90,1] + -19.628;
   1:  PR[91,2] = PR[90,2] + -20.902;
   1:  PR[91,3] = PR[90,3] + 43.452;
   1:L PR[91] R[100]mm/sec CNT100;
   1:  PR[91,1] = PR[90,1] + -16.062;
   1:  PR[91,2] = PR[90,2] + -20.868;
   1:  PR[91,3] = PR[90,3] + 43.455;
   1:L PR[91] R[100]mm/sec CNT100;
   1:  PR[91,1] = PR[90,1] + -15.690;
   1:  PR[91,2] = PR[90,2] + -20.815;
   1:  PR[91,3] = PR[90,3] + 43.465;
   1:L PR[91] R[100]mm/sec CNT100;
   1:  PR[91,1] = PR[90,1] + -11.512;
   1:  PR[91,2] = PR[90,2] + -19.887;
   1:  PR[91,3] = PR[90,3] + 43.466;
   1:L PR[91] R[100]mm/sec CNT100;
   1:  PR[91,1] = PR[90,1] + -10.372;
   1:  PR[91,2] = PR[90,2] + -19.458;
   1:  PR[91,3] = PR[90,3] + 43.478;
   1:L PR[91] R[100]mm/sec CNT100;
   1:  PR[91,1] = PR[90,1] + -7.221;
   1:  PR[91,2] = PR[90,2] + -17.999;
   1:  PR[91,3] = PR[90,3] + 43.482;
   1:L PR[91] R[100]mm/sec CNT100;
   1:  PR[91,1] = PR[90,1] + -5.510;
   1:  PR[91,2] = PR[90,2] + -16.869;
   1:  PR[91,3] = PR[90,3] + 43.492;
   1:L PR[91] R[100]mm/sec CNT100;
   1:  PR[91,1] = PR[90,1] + -3.399;
   1:  PR[91,2] = PR[90,2] + -15.246;
   1:  PR[91,3] = PR[90,3] + 43.498;
   1:L PR[91] R[100]mm/sec CNT100;
   1:  PR[91,1] = PR[90,1] + -1.479;
   1:  PR[91,2] = PR[90,2] + -13.189;
   1:  PR[91,3] = PR[90,3] + 43.505;
   1:L PR[91] R[100]mm/sec CNT100;
   1:  PR[91,1] = PR[90,1] + -0.245;
   1:  PR[91,2] = PR[90,2] + -11.676;
   1:  PR[91,3] = PR[90,3] + 43.513;
   1:L PR[91] R[100]mm/sec CNT100;
   1:  PR[91,1] = PR[90,1] + -0.231;
   1:  PR[91,2] = PR[90,2] + -11.653;
   1:  PR[91,3] = PR[90,3] + 43.519;
   1:L PR[91] R[100]mm/sec CNT100;
   1:  PR[91,1] = PR[90,1] + 2.484;
   1:  PR[91,2] = PR[90,2] + -6.464;
   1:L PR[91] R[100]mm/sec CNT100;
   1:  PR[91,1] = PR[90,1] + 5.110;
   1:  PR[91,2] = PR[90,2] + -11.698;
   1:  PR[91,3] = PR[90,3] + 43.536;
   1:L PR[91] R[100]mm/sec CNT100;
   1:  PR[91,1] = PR[90,1] + 6.021;
   1:  PR[91,2] = PR[90,2] + -12.876;
   1:  PR[91,3] = PR[90,3] + 43.552;
   1:L PR[91] R[100]mm/sec CNT100;
   1:  PR[91,1] = PR[90,1] + 7.013;
   1:  PR[91,2] = PR[90,2] + -14.304;
   1:  PR[91,3] = PR[90,3] + 43.557;
   1:L PR[91] R[100]mm/sec CNT100;
   1:  PR[91,1] = PR[90,1] + 9.158;
   1:  PR[91,2] = PR[90,2] + -16.563;
   1:  PR[91,3] = PR[90,3] + 43.562;
   1:L PR[91] R[100]mm/sec CNT100;
   1:  PR[91,1] = PR[90,1] + 11.074;
   1:  PR[91,2] = PR[90,2] + -18.017;
   1:  PR[91,3] = PR[90,3] + 43.571;
   1:L PR[91] R[100]mm/sec CNT100;
   1:  PR[91,1] = PR[90,1] + 13.593;
   1:  PR[91,2] = PR[90,2] + -19.587;
   1:  PR[91,3] = PR[90,3] + 43.577;
   1:L PR[91] R[100]mm/sec CNT100;
   1:  PR[91,1] = PR[90,1] + 15.972;
   1:  PR[91,2] = PR[90,2] + -20.558;
   1:  PR[91,3] = PR[90,3] + 43.586;
   1:L PR[91] R[100]mm/sec CNT100;
   1:  PR[91,1] = PR[90,1] + 18.642;
   1:  PR[91,2] = PR[90,2] + -21.404;
   1:  PR[91,3] = PR[90,3] + 43.593;
   1:L PR[91] R[100]mm/sec CNT100;
   1:  PR[91,1] = PR[90,1] + 21.367;
   1:  PR[91,2] = PR[90,2] + -21.753;
   1:  PR[91,3] = PR[90,3] + 43.601;
   1:L PR[91] R[100]mm/sec CNT100;
   1:  PR[91,1] = PR[90,1] + 23.983;
   1:  PR[91,2] = PR[90,2] + -21.903;
   1:  PR[91,3] = PR[90,3] + 43.609;
   1:L PR[91] R[100]mm/sec CNT100;
   1:  PR[91,1] = PR[90,1] + 26.882;
   1:  PR[91,2] = PR[90,2] + -21.517;
   1:  PR[91,3] = PR[90,3] + 43.617;
   1:L PR[91] R[100]mm/sec CNT100;
   1:  PR[91,1] = PR[90,1] + 29.278;
   1:  PR[91,2] = PR[90,2] + -21.053;
   1:  PR[91,3] = PR[90,3] + 43.625;
   1:L PR[91] R[100]mm/sec CNT100;
   1:  PR[91,1] = PR[90,1] + 32.135;
   1:  PR[91,2] = PR[90,2] + -19.875;
   1:  PR[91,3] = PR[90,3] + 43.632;
   1:L PR[91] R[100]mm/sec CNT100;
   1:  PR[91,1] = PR[90,1] + 34.191;
   1:  PR[91,2] = PR[90,2] + -18.909;
   1:  PR[91,3] = PR[90,3] + 43.641;
   1:L PR[91] R[100]mm/sec CNT100;
   1:  PR[91,1] = PR[90,1] + 36.911;
   1:  PR[91,2] = PR[90,2] + -16.845;
   1:  PR[91,3] = PR[90,3] + 43.647;
   1:L PR[91] R[100]mm/sec CNT100;
   1:  PR[91,1] = PR[90,1] + 37.156;
   1:  PR[91,2] = PR[90,2] + -16.710;
   1:  PR[91,3] = PR[90,3] + 43.657;
   1:L PR[91] R[100]mm/sec CNT100;
   1:  PR[91,1] = PR[90,1] + 37.328;
   1:  PR[91,2] = PR[90,2] + -16.593;
   1:  PR[91,3] = PR[90,3] + 43.658;
   1:L PR[91] R[100]mm/sec CNT100;
   1:  PR[91,1] = PR[90,1] + 38.729;
   1:  PR[91,2] = PR[90,2] + -15.292;
   1:L PR[91] R[100]mm/sec CNT100;
   1:  PR[91,1] = PR[90,1] + 40.034;
   1:  PR[91,2] = PR[90,2] + -13.863;
   1:  PR[91,3] = PR[90,3] + 43.664;
   1:L PR[91] R[100]mm/sec CNT100;
   1:  PR[91,1] = PR[90,1] + 43.011;
   1:  PR[91,2] = PR[90,2] + -15.658;
   1:  PR[91,3] = PR[90,3] + 43.669;
   1:L PR[91] R[100]mm/sec CNT100;
   1:  PR[91,1] = PR[90,1] + 45.519;
   1:  PR[91,2] = PR[90,2] + -17.449;
   1:  PR[91,3] = PR[90,3] + 43.679;
   1:L PR[91] R[100]mm/sec CNT100;
   1:  PR[91,1] = PR[90,1] + 46.818;
   1:  PR[91,2] = PR[90,2] + -18.299;
   1:  PR[91,3] = PR[90,3] + 43.688;
   1:L PR[91] R[100]mm/sec CNT100;
   1:  PR[91,1] = PR[90,1] + 49.353;
   1:  PR[91,2] = PR[90,2] + -19.364;
   1:  PR[91,3] = PR[90,3] + 43.693;
   1:L PR[91] R[100]mm/sec CNT100;
   1:  PR[91,1] = PR[90,1] + 53.431;
   1:  PR[91,2] = PR[90,2] + -20.937;
   1:  PR[91,3] = PR[90,3] + 43.700;
   1:L PR[91] R[100]mm/sec CNT100;
   1:  PR[91,1] = PR[90,1] + 53.830;
   1:  PR[91,2] = PR[90,2] + -21.013;
   1:  PR[91,3] = PR[90,3] + 43.713;
   1:L PR[91] R[100]mm/sec CNT100;
   1:  PR[91,1] = PR[90,1] + 58.422;
   1:  PR[91,2] = PR[90,2] + -21.990;
   1:  PR[91,3] = PR[90,3] + 43.714;
   1:L PR[91] R[100]mm/sec CNT100;
   1:  PR[91,1] = PR[90,1] + 60.850;
   1:  PR[91,2] = PR[90,2] + -22.263;
   1:  PR[91,3] = PR[90,3] + 43.728;
   1:L PR[91] R[100]mm/sec CNT100;
   1:  PR[91,1] = PR[90,1] + 63.425;
   1:  PR[91,2] = PR[90,2] + -22.308;
   1:  PR[91,3] = PR[90,3] + 43.735;
   1:L PR[91] R[100]mm/sec CNT100;
   1:  PR[91,1] = PR[90,1] + 68.513;
   1:  PR[91,2] = PR[90,2] + -21.845;
   1:  PR[91,3] = PR[90,3] + 43.742;
   1:L PR[91] R[100]mm/sec CNT100;
   1:  PR[91,1] = PR[90,1] + 68.652;
   1:  PR[91,2] = PR[90,2] + -21.821;
   1:  PR[91,3] = PR[90,3] + 43.757;
   1:L PR[91] R[100]mm/sec CNT100;
   1:  PR[91,1] = PR[90,1] + 73.536;
   1:  PR[91,2] = PR[90,2] + -20.381;
   1:L PR[91] R[100]mm/sec CNT100;
   1:  PR[91,1] = PR[90,1] + 74.427;
   1:  PR[91,2] = PR[90,2] + -20.041;
   1:  PR[91,3] = PR[90,3] + 43.771;
   1:L PR[91] R[100]mm/sec CNT100;
   1:  PR[91,1] = PR[90,1] + 77.646;
   1:  PR[91,2] = PR[90,2] + -18.262;
   1:  PR[91,3] = PR[90,3] + 43.774;
   1:L PR[91] R[100]mm/sec CNT100;
   1:  PR[91,1] = PR[90,1] + 79.302;
   1:  PR[91,2] = PR[90,2] + -17.200;
   1:  PR[91,3] = PR[90,3] + 43.785;
   1:L PR[91] R[100]mm/sec CNT100;
   1:  PR[91,1] = PR[90,1] + 81.185;
   1:  PR[91,2] = PR[90,2] + -15.519;
   1:  PR[91,3] = PR[90,3] + 43.790;
   1:L PR[91] R[100]mm/sec CNT100;
   1:  PR[91,1] = PR[90,1] + 83.084;
   1:  PR[91,2] = PR[90,2] + -13.639;
   1:  PR[91,3] = PR[90,3] + 43.798;
   1:L PR[91] R[100]mm/sec CNT100;
   1:  PR[91,1] = PR[90,1] + 84.067;
   1:  PR[91,2] = PR[90,2] + -12.229;
   1:  PR[91,3] = PR[90,3] + 43.805;
   1:L PR[91] R[100]mm/sec CNT100;
   1:  PR[91,1] = PR[90,1] + 85.771;
   1:  PR[91,2] = PR[90,2] + -9.588;
   1:  PR[91,3] = PR[90,3] + 43.810;
   1:L PR[91] R[100]mm/sec CNT100;
   1:  PR[91,1] = PR[90,1] + 86.202;
   1:  PR[91,2] = PR[90,2] + -8.472;
   1:  PR[91,3] = PR[90,3] + 43.819;
   1:L PR[91] R[100]mm/sec CNT100;
   1:  PR[91,1] = PR[90,1] + 87.371;
   1:  PR[91,2] = PR[90,2] + -5.239;
   1:  PR[91,3] = PR[90,3] + 43.822;
   1:L PR[91] R[100]mm/sec CNT100;
   1:  PR[91,1] = PR[90,1] + 87.817;
   1:  PR[91,2] = PR[90,2] + -1.463;
   1:  PR[91,3] = PR[90,3] + 43.832;
   1:L PR[91] R[100]mm/sec CNT100;
   1:  PR[91,1] = PR[90,1] + 87.945;
   1:  PR[91,2] = PR[90,2] + -0.885;
   1:  PR[91,3] = PR[90,3] + 43.843;
   1:L PR[91] R[100]mm/sec CNT100;
   1:  PR[91,1] = PR[90,1] + 87.963;
   1:  PR[91,2] = PR[90,2] + -0.736;
   1:  PR[91,3] = PR[90,3] + 43.845;
   1:L PR[91] R[100]mm/sec CNT100;
   1:  PR[91,1] = PR[90,1] + 87.376;
   1:  PR[91,2] = PR[90,2] + 3.768;
   1:L PR[91] R[100]mm/sec CNT100;
   1:  PR[91,1] = PR[90,1] + 86.202;
   1:  PR[91,2] = PR[90,2] + 7.013;
   1:  PR[91,3] = PR[90,3] + 43.858;
   1:L PR[91] R[100]mm/sec CNT100;
   1:  PR[91,1] = PR[90,1] + 85.771;
   1:  PR[91,2] = PR[90,2] + 8.129;
   1:  PR[91,3] = PR[90,3] + 43.868;
   1:L PR[91] R[100]mm/sec CNT100;
   1:  PR[91,1] = PR[90,1] + 84.067;
   1:  PR[91,2] = PR[90,2] + 10.771;
   1:  PR[91,3] = PR[90,3] + 43.872;
   1:L PR[91] R[100]mm/sec CNT100;
   1:  PR[91,1] = PR[90,1] + 83.084;
   1:  PR[91,2] = PR[90,2] + 12.181;
   1:  PR[91,3] = PR[90,3] + 43.881;
   1:L PR[91] R[100]mm/sec CNT100;
   1:  PR[91,1] = PR[90,1] + 81.185;
   1:  PR[91,2] = PR[90,2] + 14.060;
   1:  PR[91,3] = PR[90,3] + 43.885;
   1:L PR[91] R[100]mm/sec CNT100;
   1:  PR[91,1] = PR[90,1] + 79.303;
   1:  PR[91,2] = PR[90,2] + 15.741;
   1:  PR[91,3] = PR[90,3] + 43.893;
   1:L PR[91] R[100]mm/sec CNT100;
   1:  PR[91,1] = PR[90,1] + 77.646;
   1:  PR[91,2] = PR[90,2] + 16.803;
   1:  PR[91,3] = PR[90,3] + 43.900;
   1:L PR[91] R[100]mm/sec CNT100;
   1:  PR[91,1] = PR[90,1] + 74.427;
   1:  PR[91,2] = PR[90,2] + 18.582;
   1:  PR[91,3] = PR[90,3] + 43.906;
   1:L PR[91] R[100]mm/sec CNT100;
   1:  PR[91,1] = PR[90,1] + 73.537;
   1:  PR[91,2] = PR[90,2] + 18.922;
   1:  PR[91,3] = PR[90,3] + 43.916;
   1:L PR[91] R[100]mm/sec CNT100;
   1:  PR[91,1] = PR[90,1] + 68.652;
   1:  PR[91,2] = PR[90,2] + 20.362;
   1:  PR[91,3] = PR[90,3] + 43.919;
   1:L PR[91] R[100]mm/sec CNT100;
   1:  PR[91,1] = PR[90,1] + 68.511;
   1:  PR[91,2] = PR[90,2] + 20.387;
   1:  PR[91,3] = PR[90,3] + 43.934;
   1:L PR[91] R[100]mm/sec CNT100;
   1:  PR[91,1] = PR[90,1] + 63.407;
   1:  PR[91,2] = PR[90,2] + 20.851;
   1:L PR[91] R[100]mm/sec CNT100;
   1:  PR[91,1] = PR[90,1] + 60.798;
   1:  PR[91,2] = PR[90,2] + 20.799;
   1:  PR[91,3] = PR[90,3] + 43.949;
   1:L PR[91] R[100]mm/sec CNT100;
   1:  PR[91,1] = PR[90,1] + 58.380;
   1:  PR[91,2] = PR[90,2] + 20.527;
   1:  PR[91,3] = PR[90,3] + 43.956;
   1:L PR[91] R[100]mm/sec CNT100;
   1:  PR[91,1] = PR[90,1] + 53.834;
   1:  PR[91,2] = PR[90,2] + 19.546;
   1:  PR[91,3] = PR[90,3] + 43.963;
   1:L PR[91] R[100]mm/sec CNT100;
   1:  PR[91,1] = PR[90,1] + 53.338;
   1:  PR[91,2] = PR[90,2] + 19.452;
   1:  PR[91,3] = PR[90,3] + 43.976;
   1:L PR[91] R[100]mm/sec CNT100;
   1:  PR[91,1] = PR[90,1] + 49.323;
   1:  PR[91,2] = PR[90,2] + 17.884;
   1:  PR[91,3] = PR[90,3] + 43.978;
   1:L PR[91] R[100]mm/sec CNT100;
   1:  PR[91,1] = PR[90,1] + 46.809;
   1:  PR[91,2] = PR[90,2] + 16.835;
   1:  PR[91,3] = PR[90,3] + 43.990;
   1:L PR[91] R[100]mm/sec CNT100;
   1:  PR[91,1] = PR[90,1] + 45.525;
   1:  PR[91,2] = PR[90,2] + 15.987;
   1:  PR[91,3] = PR[90,3] + 43.998;
   1:L PR[91] R[100]mm/sec CNT100;
   1:  PR[91,1] = PR[90,1] + 43.009;
   1:  PR[91,2] = PR[90,2] + 14.198;
   1:  PR[91,3] = PR[90,3] + 44.002;
   1:L PR[91] R[100]mm/sec CNT100;
   1:  PR[91,1] = PR[90,1] + 40.107;
   1:  PR[91,2] = PR[90,2] + 12.371;
   1:  PR[91,3] = PR[90,3] + 44.011;
   1:L PR[91] R[100]mm/sec CNT100;
   1:  PR[91,1] = PR[90,1] + 37.247;
   1:  PR[91,2] = PR[90,2] + 15.206;
   1:  PR[91,3] = PR[90,3] + 44.021;
   1:L PR[91] R[100]mm/sec CNT100;
   1:  PR[91,1] = PR[90,1] + 35.257;
   1:  PR[91,2] = PR[90,2] + 16.711;
   1:  PR[91,3] = PR[90,3] + 44.033;
   1:L PR[91] R[100]mm/sec CNT100;
   1:  PR[91,1] = PR[90,1] + 34.502;
   1:  PR[91,2] = PR[90,2] + 17.255;
   1:  PR[91,3] = PR[90,3] + 44.040;
   1:L PR[91] R[100]mm/sec CNT100;
   1:  PR[91,1] = PR[90,1] + 34.227;
   1:  PR[91,2] = PR[90,2] + 17.436;
   1:  PR[91,3] = PR[90,3] + 44.042;
   1:L PR[91] R[100]mm/sec CNT100;
   1:  PR[91,1] = PR[90,1] + 32.113;
   1:  PR[91,2] = PR[90,2] + 18.429;
   1:  PR[91,3] = PR[90,3] + 44.043;
   1:L PR[91] R[100]mm/sec CNT100;
   1:  PR[91,1] = PR[90,1] + 29.259;
   1:  PR[91,2] = PR[90,2] + 19.599;
   1:  PR[91,3] = PR[90,3] + 44.050;
   1:L PR[91] R[100]mm/sec CNT100;
   1:  PR[91,1] = PR[90,1] + 26.863;
   1:  PR[91,2] = PR[90,2] + 20.064;
   1:  PR[91,3] = PR[90,3] + 44.059;
   1:L PR[91] R[100]mm/sec CNT100;
   1:  PR[91,1] = PR[90,1] + 23.968;
   1:  PR[91,2] = PR[90,2] + 20.444;
   1:  PR[91,3] = PR[90,3] + 44.066;
   1:L PR[91] R[100]mm/sec CNT100;
   1:  PR[91,1] = PR[90,1] + 21.354;
   1:  PR[91,2] = PR[90,2] + 20.295;
   1:  PR[91,3] = PR[90,3] + 44.074;
   1:L PR[91] R[100]mm/sec CNT100;
   1:  PR[91,1] = PR[90,1] + 18.633;
   1:  PR[91,2] = PR[90,2] + 19.942;
   1:  PR[91,3] = PR[90,3] + 44.082;
   1:L PR[91] R[100]mm/sec CNT100;
   1:  PR[91,1] = PR[90,1] + 15.964;
   1:  PR[91,2] = PR[90,2] + 19.098;
   1:  PR[91,3] = PR[90,3] + 44.089;
   1:L PR[91] R[100]mm/sec CNT100;
   1:  PR[91,1] = PR[90,1] + 13.589;
   1:  PR[91,2] = PR[90,2] + 18.126;
   1:  PR[91,3] = PR[90,3] + 44.097;
   1:L PR[91] R[100]mm/sec CNT100;
   1:  PR[91,1] = PR[90,1] + 11.071;
   1:  PR[91,2] = PR[90,2] + 16.557;
   1:  PR[91,3] = PR[90,3] + 44.105;
   1:L PR[91] R[100]mm/sec CNT100;
   1:  PR[91,1] = PR[90,1] + 9.158;
   1:  PR[91,2] = PR[90,2] + 15.104;
   1:  PR[91,3] = PR[90,3] + 44.113;
   1:L PR[91] R[100]mm/sec CNT100;
   1:  PR[91,1] = PR[90,1] + 6.978;
   1:  PR[91,2] = PR[90,2] + 12.811;
   1:  PR[91,3] = PR[90,3] + 44.120;
   1:L PR[91] R[100]mm/sec CNT100;
   1:  PR[91,1] = PR[90,1] + 5.576;
   1:  PR[91,2] = PR[90,2] + 10.998;
   1:  PR[91,3] = PR[90,3] + 44.129;
   1:L PR[91] R[100]mm/sec CNT100;
   1:  PR[91,1] = PR[90,1] + 5.270;
   1:  PR[91,2] = PR[90,2] + 10.523;
   1:  PR[91,3] = PR[90,3] + 44.136;
   1:L PR[91] R[100]mm/sec CNT100;
   1:  PR[91,1] = PR[90,1] + 2.471;
   1:  PR[91,2] = PR[90,2] + 5.173;
   1:  PR[91,3] = PR[90,3] + 44.137;
   1:L PR[91] R[100]mm/sec CNT100;
   1:  PR[91,1] = PR[90,1] + -0.258;
   1:  PR[91,2] = PR[90,2] + 10.228;
   1:  PR[91,3] = PR[90,3] + 44.155;
   1:L PR[91] R[100]mm/sec CNT100;
   1:  PR[91,1] = PR[90,1] + -1.454;
   1:  PR[91,2] = PR[90,2] + 11.697;
   1:  PR[91,3] = PR[90,3] + 44.171;
   1:L PR[91] R[100]mm/sec CNT100;
   1:  PR[91,1] = PR[90,1] + -3.383;
   1:  PR[91,2] = PR[90,2] + 13.774;
   1:  PR[91,3] = PR[90,3] + 44.176;
   1:L PR[91] R[100]mm/sec CNT100;
   1:  PR[91,1] = PR[90,1] + -5.491;
   1:  PR[91,2] = PR[90,2] + 15.396;
   1:  PR[91,3] = PR[90,3] + 44.185;
   1:L PR[91] R[100]mm/sec CNT100;
   1:  PR[91,1] = PR[90,1] + -7.203;
   1:  PR[91,2] = PR[90,2] + 16.530;
   1:  PR[91,3] = PR[90,3] + 44.192;
   1:L PR[91] R[100]mm/sec CNT100;
   1:  PR[91,1] = PR[90,1] + -10.351;
   1:  PR[91,2] = PR[90,2] + 17.991;
   1:  PR[91,3] = PR[90,3] + 44.198;
   1:L PR[91] R[100]mm/sec CNT100;
   1:  PR[91,1] = PR[90,1] + -11.495;
   1:  PR[91,2] = PR[90,2] + 18.423;
   1:  PR[91,3] = PR[90,3] + 44.208;
   1:L PR[91] R[100]mm/sec CNT100;
   1:  PR[91,1] = PR[90,1] + -15.671;
   1:  PR[91,2] = PR[90,2] + 19.353;
   1:  PR[91,3] = PR[90,3] + 44.211;
   1:L PR[91] R[100]mm/sec CNT100;
   1:  PR[91,1] = PR[90,1] + -16.046;
   1:  PR[91,2] = PR[90,2] + 19.408;
   1:  PR[91,3] = PR[90,3] + 44.224;
   1:L PR[91] R[100]mm/sec CNT100;
   1:  PR[91,1] = PR[90,1] + -19.629;
   1:  PR[91,2] = PR[90,2] + 19.444;
   1:  PR[91,3] = PR[90,3] + 44.225;
   1:L PR[91] R[100]mm/sec CNT100;
   1:  PR[91,1] = PR[90,1] + -20.787;
   1:  PR[91,2] = PR[90,2] + 19.472;
   1:  PR[91,3] = PR[90,3] + 44.235;
   1:L PR[91] R[100]mm/sec CNT100;
   1:  PR[91,1] = PR[90,1] + -25.232;
   1:  PR[91,2] = PR[90,2] + 18.617;
   1:  PR[91,3] = PR[90,3] + 44.238;
   1:L PR[91] R[100]mm/sec CNT100;
   1:  PR[91,1] = PR[90,1] + -25.716;
   1:  PR[91,2] = PR[90,2] + 18.440;
   1:  PR[91,3] = PR[90,3] + 44.251;
   1:L PR[91] R[100]mm/sec CNT100;
   1:  PR[91,1] = PR[90,1] + -29.363;
   1:  PR[91,2] = PR[90,2] + 16.881;
   1:  PR[91,3] = PR[90,3] + 44.253;
   1:L PR[91] R[100]mm/sec CNT100;
   1:  PR[91,1] = PR[90,1] + -30.199;
   1:  PR[91,2] = PR[90,2] + 16.348;
   1:  PR[91,3] = PR[90,3] + 44.264;
   1:L PR[91] R[100]mm/sec CNT100;
   1:  PR[91,1] = PR[90,1] + -33.012;
   1:  PR[91,2] = PR[90,2] + 14.344;
   1:  PR[91,3] = PR[90,3] + 44.267;
   1:L PR[91] R[100]mm/sec CNT100;
   1:  PR[91,1] = PR[90,1] + -33.977;
   1:  PR[91,2] = PR[90,2] + 13.376;
   1:  PR[91,3] = PR[90,3] + 44.277;
   1:L PR[91] R[100]mm/sec CNT100;
   1:  PR[91,1] = PR[90,1] + -36.023;
   1:  PR[91,2] = PR[90,2] + 11.114;
   1:  PR[91,3] = PR[90,3] + 44.281;
   1:L PR[91] R[100]mm/sec CNT100;
   1:  PR[91,1] = PR[90,1] + -36.985;
   1:  PR[91,2] = PR[90,2] + 9.587;
   1:  PR[91,3] = PR[90,3] + 44.289;
   1:L PR[91] R[100]mm/sec CNT100;
   1:  PR[91,1] = PR[90,1] + -37.319;
   1:  PR[91,2] = PR[90,2] + 9.182;
   1:  PR[91,3] = PR[90,3] + 44.295;
   1:L PR[91] R[100]mm/sec CNT100;
   1:  PR[91,1] = PR[90,1] + -37.860;
   1:  PR[91,2] = PR[90,2] + 8.357;
   1:  PR[91,3] = PR[90,3] + 44.296;
   1:L PR[91] R[100]mm/sec CNT100;
   1:  PR[91,1] = PR[90,1] + -39.751;
   1:  PR[91,2] = PR[90,2] + 4.692;
   1:  PR[91,3] = PR[90,3] + 44.299;
   1:L PR[91] R[100]mm/sec CNT100;
   1:  PR[91,1] = PR[90,1] + -42.239;
   1:  PR[91,2] = PR[90,2] + 7.643;
   1:  PR[91,3] = PR[90,3] + 44.311;
   1:L PR[91] R[100]mm/sec CNT100;
   1:  PR[91,1] = PR[90,1] + -44.360;
   1:  PR[91,2] = PR[90,2] + 10.554;
   1:  PR[91,3] = PR[90,3] + 44.322;
   1:L PR[91] R[100]mm/sec CNT100;
   1:  PR[91,1] = PR[90,1] + -44.909;
   1:  PR[91,2] = PR[90,2] + 11.227;
   1:  PR[91,3] = PR[90,3] + 44.332;
   1:L PR[91] R[100]mm/sec CNT100;
   1:  PR[91,1] = PR[90,1] + -47.210;
   1:  PR[91,2] = PR[90,2] + 13.172;
   1:  PR[91,3] = PR[90,3] + 44.334;
   1:L PR[91] R[100]mm/sec CNT100;
   1:  PR[91,1] = PR[90,1] + -49.243;
   1:  PR[91,2] = PR[90,2] + 14.746;
   1:  PR[91,3] = PR[90,3] + 44.343;
   1:L PR[91] R[100]mm/sec CNT100;
   1:  PR[91,1] = PR[90,1] + -50.418;
   1:  PR[91,2] = PR[90,2] + 15.369;
   1:  PR[91,3] = PR[90,3] + 44.350;
   1:L PR[91] R[100]mm/sec CNT100;
   1:  PR[91,1] = PR[90,1] + -53.729;
   1:  PR[91,2] = PR[90,2] + 16.988;
   1:  PR[91,3] = PR[90,3] + 44.354;
   1:L PR[91] R[100]mm/sec CNT100;
   1:  PR[91,1] = PR[90,1] + -54.301;
   1:  PR[91,2] = PR[90,2] + 17.299;
   1:  PR[91,3] = PR[90,3] + 44.365;
   1:L PR[91] R[100]mm/sec CNT100;
   1:  PR[91,1] = PR[90,1] + -59.056;
   1:  PR[91,2] = PR[90,2] + 18.791;
   1:  PR[91,3] = PR[90,3] + 44.367;
   1:L PR[91] R[100]mm/sec CNT100;
   1:  PR[91,1] = PR[90,1] + -61.599;
   1:  PR[91,2] = PR[90,2] + 19.113;
   1:  PR[91,3] = PR[90,3] + 44.381;
   1:L PR[91] R[100]mm/sec CNT100;
   1:  PR[91,1] = PR[90,1] + -63.981;
   1:  PR[91,2] = PR[90,2] + 19.394;
   1:  PR[91,3] = PR[90,3] + 44.388;
   1:L PR[91] R[100]mm/sec CNT100;
   1:  PR[91] = PR[90];
   1:  PR[91,1] = PR[90,1] + -66.680;
   1:  PR[91,2] = PR[90,2] + 19.362;
   1:  PR[91,3] = PR[90,3] + 45.695;
   1:L PR[91] R[100]mm/sec CNT100;
   1:  PR[91,1] = PR[90,1] + -68.182;
   1:  PR[91,2] = PR[90,2] + 19.266;
   1:  PR[91,3] = PR[90,3] + 44.405;
   1:L PR[91] R[100]mm/sec CNT100;
   1:  PR[91,1] = PR[90,1] + -72.848;
   1:  PR[91,2] = PR[90,2] + 18.145;
   1:  PR[91,3] = PR[90,3] + 44.409;
   1:L PR[91] R[100]mm/sec CNT100;
   1:  PR[91,1] = PR[90,1] + -76.898;
   1:  PR[91,2] = PR[90,2] + 16.287;
   1:  PR[91,3] = PR[90,3] + 44.423;
   1:L PR[91] R[100]mm/sec CNT100;
   1:  PR[91,1] = PR[90,1] + -77.638;
   1:  PR[91,2] = PR[90,2] + 15.760;
   1:  PR[91,3] = PR[90,3] + 44.436;
   1:L PR[91] R[100]mm/sec CNT100;
   1:  PR[91,1] = PR[90,1] + -80.414;
   1:  PR[91,2] = PR[90,2] + 13.752;
   1:  PR[91,3] = PR[90,3] + 44.439;
   1:L PR[91] R[100]mm/sec CNT100;
   1:  PR[91,1] = PR[90,1] + -83.284;
   1:  PR[91,2] = PR[90,2] + 10.642;
   1:  PR[91,3] = PR[90,3] + 44.449;
   1:L PR[91] R[100]mm/sec CNT100;
   1:  PR[91,1] = PR[90,1] + -85.404;
   1:  PR[91,2] = PR[90,2] + 7.098;
   1:  PR[91,3] = PR[90,3] + 44.461;
   1:L PR[91] R[100]mm/sec CNT100;
   1:  PR[91,1] = PR[90,1] + -86.702;
   1:  PR[91,2] = PR[90,2] + 3.258;
   1:  PR[91,3] = PR[90,3] + 44.473;
   1:L PR[91] R[100]mm/sec CNT100;
   1:  PR[91,1] = PR[90,1] + -86.984;
   1:  PR[91,2] = PR[90,2] + 0.709;
   1:  PR[91,3] = PR[90,3] + 44.485;
   1:L PR[91] R[100]mm/sec CNT100;
   1:  PR[91,1] = PR[90,1] + -87.262;
   1:  PR[91,2] = PR[90,2] + -0.734;
   1:  PR[91,3] = PR[90,3] + 44.492;
   1:L PR[91] R[100]mm/sec CNT100;
   1:  PR[91,1] = PR[90,1] + -86.843;
   1:  PR[91,2] = PR[90,2] + -4.504;
   1:  PR[91,3] = PR[90,3] + 44.496;
   1:L PR[91] R[100]mm/sec CNT100;
   1:  PR[91,1] = PR[90,1] + -86.818;
   1:  PR[91,2] = PR[90,2] + -4.671;
   1:  PR[91,3] = PR[90,3] + 44.507;
   1:L PR[91] R[100]mm/sec CNT100;
   1:  PR[91,1] = PR[90,1] + -85.555;
   1:  PR[91,2] = PR[90,2] + -8.344;
   1:  PR[91,3] = PR[90,3] + 44.508;
   1:L PR[91] R[100]mm/sec CNT100;
   1:  PR[91,1] = PR[90,1] + -85.487;
   1:  PR[91,2] = PR[90,2] + -8.545;
   1:  PR[91,3] = PR[90,3] + 44.519;
   1:L PR[91] R[100]mm/sec CNT100;
   1:  PR[91,1] = PR[90,1] + -83.335;
   1:  PR[91,2] = PR[90,2] + -12.085;
   1:  PR[91,3] = PR[90,3] + 44.520;
   1:L PR[91] R[100]mm/sec CNT100;
   1:  PR[91,1] = PR[90,1] + -80.418;
   1:  PR[91,2] = PR[90,2] + -15.197;
   1:  PR[91,3] = PR[90,3] + 44.532;
   1:L PR[91] R[100]mm/sec CNT100;
   1:  PR[91,1] = PR[90,1] + -78.082;
   1:  PR[91,2] = PR[90,2] + -16.842;
   1:  PR[91,3] = PR[90,3] + 44.544;
   1:L PR[91] R[100]mm/sec CNT100;
   1:  PR[91,1] = PR[90,1] + -76.824;
   1:  PR[91,2] = PR[90,2] + -17.751;
   1:  PR[91,3] = PR[90,3] + 44.553;
   1:L PR[91] R[100]mm/sec CNT100;
   1:  PR[91,1] = PR[90,1] + -74.749;
   1:  PR[91,2] = PR[90,2] + -18.674;
   1:  PR[91,3] = PR[90,3] + 44.557;
   1:L PR[91] R[100]mm/sec CNT100;
   1:  PR[91,1] = PR[90,1] + -72.695;
   1:  PR[91,2] = PR[90,2] + -19.623;
   1:  PR[91,3] = PR[90,3] + 44.564;
   1:L PR[91] R[100]mm/sec CNT100;
   1:  PR[91,1] = PR[90,1] + -71.190;
   1:  PR[91,2] = PR[90,2] + -19.973;
   1:  PR[91,3] = PR[90,3] + 44.570;
   1:L PR[91] R[100]mm/sec CNT100;
   1:  PR[91,1] = PR[90,1] + -68.178;
   1:  PR[91,2] = PR[90,2] + -20.723;
   1:  PR[91,3] = PR[90,3] + 44.575;
   1:L PR[91] R[100]mm/sec CNT100;
   1:  PR[91,1] = PR[90,1] + -67.504;
   1:  PR[91,2] = PR[90,2] + -20.751;
   1:  PR[91,3] = PR[90,3] + 44.584;
   1:L PR[91] R[100]mm/sec CNT100;
   1:  PR[91,1] = PR[90,1] + -63.363;
   1:  PR[91,2] = PR[90,2] + -20.995;
   1:  PR[91,3] = PR[90,3] + 44.586;
   1:L PR[91] R[100]mm/sec CNT100;
   1:  PR[91,1] = PR[90,1] + -63.305;
   1:  PR[91,2] = PR[90,2] + -20.994;
   1:  PR[91,3] = PR[90,3] + 44.598;
   1:L PR[91] R[100]mm/sec CNT100;
   1:  PR[91,1] = PR[90,1] + -58.956;
   1:  PR[91,2] = PR[90,2] + -20.524;
   1:L PR[91] R[100]mm/sec CNT100;
   1:  PR[91,1] = PR[90,1] + -57.107;
   1:  PR[91,2] = PR[90,2] + -20.157;
   1:  PR[91,3] = PR[90,3] + 44.611;
   1:L PR[91] R[100]mm/sec CNT100;
   1:  PR[91,1] = PR[90,1] + -54.576;
   1:  PR[91,2] = PR[90,2] + -19.408;
   1:  PR[91,3] = PR[90,3] + 44.616;
   1:L PR[91] R[100]mm/sec CNT100;
   1:  PR[91,1] = PR[90,1] + -50.900;
   1:  PR[91,2] = PR[90,2] + -17.887;
   1:  PR[91,3] = PR[90,3] + 44.624;
   1:L PR[91] R[100]mm/sec CNT100;
   1:  PR[91,1] = PR[90,1] + -50.323;
   1:  PR[91,2] = PR[90,2] + -17.587;
   1:  PR[91,3] = PR[90,3] + 44.635;
   1:L PR[91] R[100]mm/sec CNT100;
   1:  PR[91,1] = PR[90,1] + -48.496;
   1:  PR[91,2] = PR[90,2] + -16.328;
   1:  PR[91,3] = PR[90,3] + 44.637;
   1:L PR[91] R[100]mm/sec CNT100;
   1:  PR[91,1] = PR[90,1] + -45.705;
   1:  PR[91,2] = PR[90,2] + -14.658;
   1:  PR[91,3] = PR[90,3] + 44.644;
   1:L PR[91] R[100]mm/sec CNT100;
   1:  PR[91,1] = PR[90,1] + -44.245;
   1:  PR[91,2] = PR[90,2] + -13.281;
   1:  PR[91,3] = PR[90,3] + 44.653;
   1:L PR[91] R[100]mm/sec CNT100;
   1:  PR[91,1] = PR[90,1] + -41.796;
   1:  PR[91,2] = PR[90,2] + -10.906;
   1:  PR[91,3] = PR[90,3] + 44.659;
   1:L PR[91] R[100]mm/sec CNT100;
   1:  PR[91,1] = PR[90,1] + -39.236;
   1:  PR[91,2] = PR[90,2] + -6.838;
   1:  PR[91,3] = PR[90,3] + 44.669;
   1:L PR[91] R[100]mm/sec CNT100;
   1:  PR[91,1] = PR[90,1] + -37.187;
   1:  PR[91,2] = PR[90,2] + -10.633;
   1:  PR[91,3] = PR[90,3] + 44.683;
   1:L PR[91] R[100]mm/sec CNT100;
   1:  PR[91,1] = PR[90,1] + -36.936;
   1:  PR[91,2] = PR[90,2] + -11.033;
   1:  PR[91,3] = PR[90,3] + 44.695;
   1:L PR[91] R[100]mm/sec CNT100;
   1:  PR[91,1] = PR[90,1] + -36.583;
   1:  PR[91,2] = PR[90,2] + -11.561;
   1:  PR[91,3] = PR[90,3] + 44.697;
   1:L PR[91] R[100]mm/sec CNT100;
   1:  PR[91,1] = PR[90,1] + -35.894;
   1:  PR[91,2] = PR[90,2] + -12.506;
   1:  PR[91,3] = PR[90,3] + 44.698;
   1:L PR[91] R[100]mm/sec CNT100;
   1:  PR[91,1] = PR[90,1] + -33.466;
   1:  PR[91,2] = PR[90,2] + -15.194;
   1:  PR[91,3] = PR[90,3] + 44.702;
   1:L PR[91] R[100]mm/sec CNT100;
   1:  PR[91,1] = PR[90,1] + -32.840;
   1:  PR[91,2] = PR[90,2] + -15.822;
   1:  PR[91,3] = PR[90,3] + 44.712;
   1:L PR[91] R[100]mm/sec CNT100;
   1:  PR[91,1] = PR[90,1] + -29.605;
   1:  PR[91,2] = PR[90,2] + -18.128;
   1:  PR[91,3] = PR[90,3] + 44.715;
   1:L PR[91] R[100]mm/sec CNT100;
   1:  PR[91,1] = PR[90,1] + -29.193;
   1:  PR[91,2] = PR[90,2] + -18.391;
   1:  PR[91,3] = PR[90,3] + 44.726;
   1:L PR[91] R[100]mm/sec CNT100;
   1:  PR[91,1] = PR[90,1] + -25.052;
   1:  PR[91,2] = PR[90,2] + -20.164;
   1:  PR[91,3] = PR[90,3] + 44.728;
   1:L PR[91] R[100]mm/sec CNT100;
   1:  PR[91,1] = PR[90,1] + -20.432;
   1:  PR[91,2] = PR[90,2] + -21.079;
   1:  PR[91,3] = PR[90,3] + 44.741;
   1:L PR[91] R[100]mm/sec CNT100;
   1:  PR[91,1] = PR[90,1] + -20.156;
   1:  PR[91,2] = PR[90,2] + -21.099;
   1:  PR[91,3] = PR[90,3] + 44.755;
   1:L PR[91] R[100]mm/sec CNT100;
   1:  PR[91,1] = PR[90,1] + -15.783;
   1:  PR[91,2] = PR[90,2] + -21.057;
   1:L PR[91] R[100]mm/sec CNT100;
   1:  PR[91,1] = PR[90,1] + -14.689;
   1:  PR[91,2] = PR[90,2] + -20.901;
   1:  PR[91,3] = PR[90,3] + 44.768;
   1:L PR[91] R[100]mm/sec CNT100;
   1:  PR[91,1] = PR[90,1] + -11.178;
   1:  PR[91,2] = PR[90,2] + -20.121;
   1:  PR[91,3] = PR[90,3] + 44.771;
   1:L PR[91] R[100]mm/sec CNT100;
   1:  PR[91,1] = PR[90,1] + -9.318;
   1:  PR[91,2] = PR[90,2] + -19.421;
   1:  PR[91,3] = PR[90,3] + 44.782;
   1:L PR[91] R[100]mm/sec CNT100;
   1:  PR[91,1] = PR[90,1] + -6.819;
   1:  PR[91,2] = PR[90,2] + -18.264;
   1:  PR[91,3] = PR[90,3] + 44.787;
   1:L PR[91] R[100]mm/sec CNT100;
   1:  PR[91,1] = PR[90,1] + -4.440;
   1:  PR[91,2] = PR[90,2] + -16.692;
   1:  PR[91,3] = PR[90,3] + 44.795;
   1:L PR[91] R[100]mm/sec CNT100;
   1:  PR[91,1] = PR[90,1] + -2.920;
   1:  PR[91,2] = PR[90,2] + -15.524;
   1:  PR[91,3] = PR[90,3] + 44.804;
   1:L PR[91] R[100]mm/sec CNT100;
   1:  PR[91,1] = PR[90,1] + -0.433;
   1:  PR[91,2] = PR[90,2] + -12.859;
   1:  PR[91,3] = PR[90,3] + 44.809;
   1:L PR[91] R[100]mm/sec CNT100;
   1:  PR[91,1] = PR[90,1] + 0.313;
   1:  PR[91,2] = PR[90,2] + -11.944;
   1:  PR[91,3] = PR[90,3] + 44.820;
   1:L PR[91] R[100]mm/sec CNT100;
   1:  PR[91,1] = PR[90,1] + 0.354;
   1:  PR[91,2] = PR[90,2] + -11.875;
   1:  PR[91,3] = PR[90,3] + 44.823;
   1:L PR[91] R[100]mm/sec CNT100;
   1:  PR[91,1] = PR[90,1] + 2.668;
   1:  PR[91,2] = PR[90,2] + -7.453;
   1:  PR[91,3] = PR[90,3] + 44.824;
   1:L PR[91] R[100]mm/sec CNT100;
   1:  PR[91,1] = PR[90,1] + 4.878;
   1:  PR[91,2] = PR[90,2] + -11.859;
   1:  PR[91,3] = PR[90,3] + 44.838;
   1:L PR[91] R[100]mm/sec CNT100;
   1:  PR[91,1] = PR[90,1] + 5.359;
   1:  PR[91,2] = PR[90,2] + -12.480;
   1:  PR[91,3] = PR[90,3] + 44.852;
   1:L PR[91] R[100]mm/sec CNT100;
   1:  PR[91,1] = PR[90,1] + 6.530;
   1:  PR[91,2] = PR[90,2] + -14.166;
   1:  PR[91,3] = PR[90,3] + 44.855;
   1:L PR[91] R[100]mm/sec CNT100;
   1:  PR[91,1] = PR[90,1] + 9.075;
   1:  PR[91,2] = PR[90,2] + -16.848;
   1:  PR[91,3] = PR[90,3] + 44.861;
   1:L PR[91] R[100]mm/sec CNT100;
   1:  PR[91,1] = PR[90,1] + 10.559;
   1:  PR[91,2] = PR[90,2] + -17.972;
   1:  PR[91,3] = PR[90,3] + 44.871;
   1:L PR[91] R[100]mm/sec CNT100;
   1:  PR[91,1] = PR[90,1] + 13.561;
   1:  PR[91,2] = PR[90,2] + -19.844;
   1:  PR[91,3] = PR[90,3] + 44.877;
   1:L PR[91] R[100]mm/sec CNT100;
   1:  PR[91,1] = PR[90,1] + 15.442;
   1:  PR[91,2] = PR[90,2] + -20.612;
   1:  PR[91,3] = PR[90,3] + 44.887;
   1:L PR[91] R[100]mm/sec CNT100;
   1:  PR[91,1] = PR[90,1] + 18.649;
   1:  PR[91,2] = PR[90,2] + -21.627;
   1:  PR[91,3] = PR[90,3] + 44.893;
   1:L PR[91] R[100]mm/sec CNT100;
   1:  PR[91,1] = PR[90,1] + 20.846;
   1:  PR[91,2] = PR[90,2] + -21.909;
   1:  PR[91,3] = PR[90,3] + 44.903;
   1:L PR[91] R[100]mm/sec CNT100;
   1:  PR[91,1] = PR[90,1] + 24.019;
   1:  PR[91,2] = PR[90,2] + -22.091;
   1:  PR[91,3] = PR[90,3] + 44.909;
   1:L PR[91] R[100]mm/sec CNT100;
   1:  PR[91,1] = PR[90,1] + 26.397;
   1:  PR[91,2] = PR[90,2] + -21.775;
   1:  PR[91,3] = PR[90,3] + 44.918;
   1:L PR[91] R[100]mm/sec CNT100;
   1:  PR[91,1] = PR[90,1] + 29.333;
   1:  PR[91,2] = PR[90,2] + -21.206;
   1:  PR[91,3] = PR[90,3] + 44.925;
   1:L PR[91] R[100]mm/sec CNT100;
   1:  PR[91,1] = PR[90,1] + 31.711;
   1:  PR[91,2] = PR[90,2] + -20.225;
   1:  PR[91,3] = PR[90,3] + 44.934;
   1:L PR[91] R[100]mm/sec CNT100;
   1:  PR[91,1] = PR[90,1] + 34.258;
   1:  PR[91,2] = PR[90,2] + -19.029;
   1:  PR[91,3] = PR[90,3] + 44.941;
   1:L PR[91] R[100]mm/sec CNT100;
   1:  PR[91,1] = PR[90,1] + 36.572;
   1:  PR[91,2] = PR[90,2] + -17.273;
   1:  PR[91,3] = PR[90,3] + 44.950;
   1:L PR[91] R[100]mm/sec CNT100;
   1:  PR[91,1] = PR[90,1] + 36.862;
   1:  PR[91,2] = PR[90,2] + -17.113;
   1:  PR[91,3] = PR[90,3] + 44.958;
   1:L PR[91] R[100]mm/sec CNT100;
   1:  PR[91,1] = PR[90,1] + 37.117;
   1:  PR[91,2] = PR[90,2] + -16.939;
   1:  PR[91,3] = PR[90,3] + 44.959;
   1:L PR[91] R[100]mm/sec CNT100;
   1:  PR[91,1] = PR[90,1] + 39.490;
   1:  PR[91,2] = PR[90,2] + -14.736;
   1:  PR[91,3] = PR[90,3] + 44.960;
   1:L PR[91] R[100]mm/sec CNT100;
   1:  PR[91,1] = PR[90,1] + 44.483;
   1:  PR[91,2] = PR[90,2] + -17.820;
   1:  PR[91,3] = PR[90,3] + 44.969;
   1:L PR[91] R[100]mm/sec CNT100;
   1:  PR[91,1] = PR[90,1] + 45.118;
   1:  PR[91,2] = PR[90,2] + -18.273;
   1:  PR[91,3] = PR[90,3] + 44.986;
   1:L PR[91] R[100]mm/sec CNT100;
   1:  PR[91,1] = PR[90,1] + 45.300;
   1:  PR[91,2] = PR[90,2] + -18.392;
   1:  PR[91,3] = PR[90,3] + 44.989;
   1:L PR[91] R[100]mm/sec CNT100;
   1:  PR[91,1] = PR[90,1] + 49.080;
   1:  PR[91,2] = PR[90,2] + -19.979;
   1:L PR[91] R[100]mm/sec CNT100;
   1:  PR[91,1] = PR[90,1] + 52.043;
   1:  PR[91,2] = PR[90,2] + -21.123;
   1:  PR[91,3] = PR[90,3] + 45.001;
   1:L PR[91] R[100]mm/sec CNT100;
   1:  PR[91,1] = PR[90,1] + 53.257;
   1:  PR[91,2] = PR[90,2] + -21.370;
   1:  PR[91,3] = PR[90,3] + 45.010;
   1:L PR[91] R[100]mm/sec CNT100;
   1:  PR[91,1] = PR[90,1] + 55.752;
   1:  PR[91,2] = PR[90,2] + -21.820;
   1:  PR[91,3] = PR[90,3] + 45.014;
   1:L PR[91] R[100]mm/sec CNT100;
   1:  PR[91,1] = PR[90,1] + 58.118;
   1:  PR[91,2] = PR[90,2] + -22.323;
   1:  PR[91,3] = PR[90,3] + 45.021;
   1:L PR[91] R[100]mm/sec CNT100;
   1:  PR[91,1] = PR[90,1] + 59.291;
   1:  PR[91,2] = PR[90,2] + -22.455;
   1:  PR[91,3] = PR[90,3] + 45.028;
   1:L PR[91] R[100]mm/sec CNT100;
   1:  PR[91,1] = PR[90,1] + 63.095;
   1:  PR[91,2] = PR[90,2] + -22.522;
   1:  PR[91,3] = PR[90,3] + 45.032;
   1:L PR[91] R[100]mm/sec CNT100;
   1:  PR[91,1] = PR[90,1] + 66.999;
   1:  PR[91,2] = PR[90,2] + -22.167;
   1:  PR[91,3] = PR[90,3] + 45.043;
   1:L PR[91] R[100]mm/sec CNT100;
   1:  PR[91,1] = PR[90,1] + 68.277;
   1:  PR[91,2] = PR[90,2] + -21.945;
   1:  PR[91,3] = PR[90,3] + 45.054;
   1:L PR[91] R[100]mm/sec CNT100;
   1:  PR[91,1] = PR[90,1] + 73.428;
   1:  PR[91,2] = PR[90,2] + -20.409;
   1:  PR[91,3] = PR[90,3] + 45.058;
   1:L PR[91] R[100]mm/sec CNT100;
   1:  PR[91,1] = PR[90,1] + 73.641;
   1:  PR[91,2] = PR[90,2] + -20.327;
   1:  PR[91,3] = PR[90,3] + 45.073;
   1:L PR[91] R[100]mm/sec CNT100;
   1:  PR[91,1] = PR[90,1] + 77.548;
   1:  PR[91,2] = PR[90,2] + -18.168;
   1:  PR[91,3] = PR[90,3] + 45.074;
   1:L PR[91] R[100]mm/sec CNT100;
   1:  PR[91,1] = PR[90,1] + 78.651;
   1:  PR[91,2] = PR[90,2] + -17.462;
   1:  PR[91,3] = PR[90,3] + 45.087;
   1:L PR[91] R[100]mm/sec CNT100;
   1:  PR[91,1] = PR[90,1] + 81.067;
   1:  PR[91,2] = PR[90,2] + -15.304;
   1:  PR[91,3] = PR[90,3] + 45.091;
   1:L PR[91] R[100]mm/sec CNT100;
   1:  PR[91,1] = PR[90,1] + 82.534;
   1:  PR[91,2] = PR[90,2] + -13.852;
   1:  PR[91,3] = PR[90,3] + 45.100;
   1:L PR[91] R[100]mm/sec CNT100;
   1:  PR[91,1] = PR[90,1] + 83.900;
   1:  PR[91,2] = PR[90,2] + -11.894;
   1:  PR[91,3] = PR[90,3] + 45.106;
   1:L PR[91] R[100]mm/sec CNT100;
   1:  PR[91,1] = PR[90,1] + 85.291;
   1:  PR[91,2] = PR[90,2] + -9.736;
   1:  PR[91,3] = PR[90,3] + 45.113;
   1:L PR[91] R[100]mm/sec CNT100;
   1:  PR[91,1] = PR[90,1] + 85.955;
   1:  PR[91,2] = PR[90,2] + -8.019;
   1:  PR[91,3] = PR[90,3] + 45.121;
   1:L PR[91] R[100]mm/sec CNT100;
   1:  PR[91,1] = PR[90,1] + 86.933;
   1:  PR[91,2] = PR[90,2] + -5.315;
   1:  PR[91,3] = PR[90,3] + 45.126;
   1:L PR[91] R[100]mm/sec CNT100;
   1:  PR[91,1] = PR[90,1] + 87.308;
   1:  PR[91,2] = PR[90,2] + -2.135;
   1:  PR[91,3] = PR[90,3] + 45.134;
   1:L PR[91] R[100]mm/sec CNT100;
   1:  PR[91,1] = PR[90,1] + 87.416;
   1:  PR[91,2] = PR[90,2] + -1.644;
   1:  PR[91,3] = PR[90,3] + 45.144;
   1:L PR[91] R[100]mm/sec CNT100;
   1:  PR[91,1] = PR[90,1] + 87.528;
   1:  PR[91,2] = PR[90,2] + -0.738;
   1:  PR[91,3] = PR[90,3] + 45.145;
   1:L PR[91] R[100]mm/sec CNT100;
   1:  PR[91,1] = PR[90,1] + 87.126;
   1:  PR[91,2] = PR[90,2] + 2.303;
   1:  PR[91,3] = PR[90,3] + 45.148;
   1:L PR[91] R[100]mm/sec CNT100;
   1:  PR[91,1] = PR[90,1] + 86.935;
   1:  PR[91,2] = PR[90,2] + 3.851;
   1:  PR[91,3] = PR[90,3] + 45.157;
   1:L PR[91] R[100]mm/sec CNT100;
   1:  PR[91,1] = PR[90,1] + 85.955;
   1:  PR[91,2] = PR[90,2] + 6.560;
   1:  PR[91,3] = PR[90,3] + 45.161;
   1:L PR[91] R[100]mm/sec CNT100;
   1:  PR[91,1] = PR[90,1] + 85.291;
   1:  PR[91,2] = PR[90,2] + 8.277;
   1:  PR[91,3] = PR[90,3] + 45.169;
   1:L PR[91] R[100]mm/sec CNT100;
   1:  PR[91,1] = PR[90,1] + 83.900;
   1:  PR[91,2] = PR[90,2] + 10.435;
   1:  PR[91,3] = PR[90,3] + 45.175;
   1:L PR[91] R[100]mm/sec CNT100;
   1:  PR[91,1] = PR[90,1] + 82.534;
   1:  PR[91,2] = PR[90,2] + 12.393;
   1:  PR[91,3] = PR[90,3] + 45.182;
   1:L PR[91] R[100]mm/sec CNT100;
   1:  PR[91,1] = PR[90,1] + 81.067;
   1:  PR[91,2] = PR[90,2] + 13.845;
   1:  PR[91,3] = PR[90,3] + 45.189;
   1:L PR[91] R[100]mm/sec CNT100;
   1:  PR[91,1] = PR[90,1] + 78.651;
   1:  PR[91,2] = PR[90,2] + 16.003;
   1:  PR[91,3] = PR[90,3] + 45.195;
   1:L PR[91] R[100]mm/sec CNT100;
   1:  PR[91,1] = PR[90,1] + 77.549;
   1:  PR[91,2] = PR[90,2] + 16.709;
   1:  PR[91,3] = PR[90,3] + 45.205;
   1:L PR[91] R[100]mm/sec CNT100;
   1:  PR[91,1] = PR[90,1] + 73.642;
   1:  PR[91,2] = PR[90,2] + 18.868;
   1:  PR[91,3] = PR[90,3] + 45.208;
   1:L PR[91] R[100]mm/sec CNT100;
   1:  PR[91,1] = PR[90,1] + 73.428;
   1:  PR[91,2] = PR[90,2] + 18.950;
   1:  PR[91,3] = PR[90,3] + 45.221;
   1:L PR[91] R[100]mm/sec CNT100;
   1:  PR[91,1] = PR[90,1] + 68.270;
   1:  PR[91,2] = PR[90,2] + 20.489;
   1:  PR[91,3] = PR[90,3] + 45.222;
   1:L PR[91] R[100]mm/sec CNT100;
   1:  PR[91,1] = PR[90,1] + 66.977;
   1:  PR[91,2] = PR[90,2] + 20.710;
   1:  PR[91,3] = PR[90,3] + 45.238;
   1:L PR[91] R[100]mm/sec CNT100;
   1:  PR[91,1] = PR[90,1] + 63.068;
   1:  PR[91,2] = PR[90,2] + 21.066;
   1:  PR[91,3] = PR[90,3] + 45.241;
   1:L PR[91] R[100]mm/sec CNT100;
   1:  PR[91,1] = PR[90,1] + 59.214;
   1:  PR[91,2] = PR[90,2] + 20.989;
   1:  PR[91,3] = PR[90,3] + 45.253;
   1:L PR[91] R[100]mm/sec CNT100;
   1:  PR[91,1] = PR[90,1] + 58.065;
   1:  PR[91,2] = PR[90,2] + 20.860;
   1:  PR[91,3] = PR[90,3] + 45.264;
   1:L PR[91] R[100]mm/sec CNT100;
   1:  PR[91,1] = PR[90,1] + 55.759;
   1:  PR[91,2] = PR[90,2] + 20.363;
   1:  PR[91,3] = PR[90,3] + 45.267;
   1:L PR[91] R[100]mm/sec CNT100;
   1:  PR[91,1] = PR[90,1] + 53.207;
   1:  PR[91,2] = PR[90,2] + 19.893;
   1:  PR[91,3] = PR[90,3] + 45.274;
   1:L PR[91] R[100]mm/sec CNT100;
   1:  PR[91,1] = PR[90,1] + 51.984;
   1:  PR[91,2] = PR[90,2] + 19.647;
   1:  PR[91,3] = PR[90,3] + 45.282;
   1:L PR[91] R[100]mm/sec CNT100;
   1:  PR[91,1] = PR[90,1] + 49.065;
   1:  PR[91,2] = PR[90,2] + 18.507;
   1:  PR[91,3] = PR[90,3] + 45.285;
   1:L PR[91] R[100]mm/sec CNT100;
   1:  PR[91,1] = PR[90,1] + 45.352;
   1:  PR[91,2] = PR[90,2] + 16.958;
   1:  PR[91,3] = PR[90,3] + 45.294;
   1:L PR[91] R[100]mm/sec CNT100;
   1:  PR[91,1] = PR[90,1] + 44.475;
   1:  PR[91,2] = PR[90,2] + 16.351;
   1:  PR[91,3] = PR[90,3] + 45.306;
   1:L PR[91] R[100]mm/sec CNT100;
   1:  PR[91,1] = PR[90,1] + 39.433;
   1:  PR[91,2] = PR[90,2] + 13.177;
   1:  PR[91,3] = PR[90,3] + 45.309;
   1:L PR[91] R[100]mm/sec CNT100;
   1:  PR[91,1] = PR[90,1] + 37.041;
   1:  PR[91,2] = PR[90,2] + 15.548;
   1:  PR[91,3] = PR[90,3] + 45.327;
   1:L PR[91] R[100]mm/sec CNT100;
   1:  PR[91,1] = PR[90,1] + 35.593;
   1:  PR[91,2] = PR[90,2] + 16.643;
   1:  PR[91,3] = PR[90,3] + 45.336;
   1:L PR[91] R[100]mm/sec CNT100;
   1:  PR[91,1] = PR[90,1] + 34.665;
   1:  PR[91,2] = PR[90,2] + 17.312;
   1:  PR[91,3] = PR[90,3] + 45.342;
   1:L PR[91] R[100]mm/sec CNT100;
   1:  PR[91,1] = PR[90,1] + 34.298;
   1:  PR[91,2] = PR[90,2] + 17.553;
   1:  PR[91,3] = PR[90,3] + 45.345;
   1:L PR[91] R[100]mm/sec CNT100;
   1:  PR[91,1] = PR[90,1] + 31.694;
   1:  PR[91,2] = PR[90,2] + 18.777;
   1:  PR[91,3] = PR[90,3] + 45.346;
   1:L PR[91] R[100]mm/sec CNT100;
   1:  PR[91,1] = PR[90,1] + 29.317;
   1:  PR[91,2] = PR[90,2] + 19.751;
   1:  PR[91,3] = PR[90,3] + 45.355;
   1:L PR[91] R[100]mm/sec CNT100;
   1:  PR[91,1] = PR[90,1] + 26.382;
   1:  PR[91,2] = PR[90,2] + 20.320;
   1:  PR[91,3] = PR[90,3] + 45.362;
   1:L PR[91] R[100]mm/sec CNT100;
   1:  PR[91,1] = PR[90,1] + 24.007;
   1:  PR[91,2] = PR[90,2] + 20.632;
   1:  PR[91,3] = PR[90,3] + 45.371;
   1:L PR[91] R[100]mm/sec CNT100;
   1:  PR[91,1] = PR[90,1] + 20.837;
   1:  PR[91,2] = PR[90,2] + 20.451;
   1:  PR[91,3] = PR[90,3] + 45.378;
   1:L PR[91] R[100]mm/sec CNT100;
   1:  PR[91,1] = PR[90,1] + 18.643;
   1:  PR[91,2] = PR[90,2] + 20.167;
   1:  PR[91,3] = PR[90,3] + 45.387;
   1:L PR[91] R[100]mm/sec CNT100;
   1:  PR[91,1] = PR[90,1] + 15.437;
   1:  PR[91,2] = PR[90,2] + 19.153;
   1:  PR[91,3] = PR[90,3] + 45.393;
   1:L PR[91] R[100]mm/sec CNT100;
   1:  PR[91,1] = PR[90,1] + 13.560;
   1:  PR[91,2] = PR[90,2] + 18.384;
   1:  PR[91,3] = PR[90,3] + 45.403;
   1:L PR[91] R[100]mm/sec CNT100;
   1:  PR[91,1] = PR[90,1] + 10.558;
   1:  PR[91,2] = PR[90,2] + 16.515;
   1:  PR[91,3] = PR[90,3] + 45.409;
   1:L PR[91] R[100]mm/sec CNT100;
   1:  PR[91,1] = PR[90,1] + 9.078;
   1:  PR[91,2] = PR[90,2] + 15.390;
   1:  PR[91,3] = PR[90,3] + 45.419;
   1:L PR[91] R[100]mm/sec CNT100;
   1:  PR[91,1] = PR[90,1] + 6.497;
   1:  PR[91,2] = PR[90,2] + 12.675;
   1:  PR[91,3] = PR[90,3] + 45.425;
   1:L PR[91] R[100]mm/sec CNT100;
   1:  PR[91,1] = PR[90,1] + 5.421;
   1:  PR[91,2] = PR[90,2] + 11.285;
   1:  PR[91,3] = PR[90,3] + 45.435;
   1:L PR[91] R[100]mm/sec CNT100;
   1:  PR[91,1] = PR[90,1] + 5.280;
   1:  PR[91,2] = PR[90,2] + 11.075;
   1:  PR[91,3] = PR[90,3] + 45.441;
   1:L PR[91] R[100]mm/sec CNT100;
   1:  PR[91,1] = PR[90,1] + 5.067;
